// TwinCAT 3 PLC project IDPLC
// ProgramVersion: 3.1.4024.12
// libraries:
//   Tc2_Drive, * (Beckhoff Automation GmbH)
//   Tc2_EtherCAT, * (Beckhoff Automation GmbH)
//   Tc2_Math, * (Beckhoff Automation GmbH)
//   Tc2_MC2, * (Beckhoff Automation GmbH)
//   Tc2_NC, * (Beckhoff Automation GmbH)
//   Tc2_NcDrive, * (Beckhoff Automation GmbH)
//   Tc2_SerialCom, * (Beckhoff Automation GmbH)
//   Tc2_Standard, * (Beckhoff Automation GmbH)
//   Tc2_System, * (Beckhoff Automation GmbH)
//   Tc2_Utilities, * (Beckhoff Automation GmbH)
//   Tc3_Module, * (Beckhoff Automation GmbH)
// project tree:
//   DUTs/ DUT_SENSOR_DATAS_1.TcDUT (not stored), DUT_SENSOR_DATAS_8.TcDUT (not stored), DUT_SENSOR_DATAS_2.TcDUT (not stored), DUT_SENSOR_DATAS_3.TcDUT (not stored), DUT_SENSOR_DATAS_4.TcDUT (not stored), DUT_SENSOR_DATAS_5.TcDUT (not stored), DUT_SENSOR_DATAS_6.TcDUT (not stored), DUT_SENSOR_DATAS_7.TcDUT (not stored), Struct_M_Compensation.TcDUT, ST_P180.TcDUT, ST_P182.TcDUT, ST_P183.TcDUT
//   GVLs/ Global_Variables.TcGVL, Variable_Configuration.TcGVL (not stored)
//   / PlcTask.TcTTO (not stored), RecipeManager.TcRMO (not stored)
//   POUs/0.UserMode/ F_GetSysTime.TcPOU (not stored), UserMode.TcPOU
//   POUs/CommonFB/ExternFB/ FB_LedShow.TcPOU (not stored), FB_PlcEmergencyStop.TcPOU (not stored)
//   POUs/CommonFB/MainFB/ FB_Move.TcPOU, FB_Power.TcPOU, FB_SetAxisPosition.TcPOU, FB_SetMotorAxisPosition.TcPOU, FB_Stop.TcPOU
//   POUs/ MAIN.TcPOU
//   POUs/RS232/ BackgroundEL.TcPOU (not stored), FB_SerialCom.TcPOU (not stored)

// ---- DUTs/Struct_M_Compensation.TcDUT
TYPE Struct_M_Compensation :
STRUCT
	Gap:LREAL;
	PhaseShifterLin:LREAL;
	InRange:BOOL;
END_STRUCT
END_TYPE

// ---- DUTs/ST_P180.TcDUT
//Feedback 2 type
TYPE ST_P180 :
STRUCT
	iActual_lenght:UINT:=224;
	iMax_lenght:UINT:=224;

	Manufacturer:UINT:=2;
	Feedback_type:UINT:=1;
	Feedback_type_string:STRING(29):='hallo';
	Feedback_use:UINT:=3;
	Feedback_direction:UINT:=1;
	(*rsvd*)
		rsvd1:ARRAY[0..2] OF UINT;

	(*Powersettlings*)
		Control_voltage:UINT;
		Wait_time_after_power_up:UINT;
		Connector:UINT;
		rsvd2:ARRAY[0..2] OF UINT;

	(*Process channel*)
		Process_interface:UINT;
		Conector2:UINT;
			(*rsvd*)
				rsvd3:ARRAY[0..1] OF UINT;
			(*Data*)
				(*Sin/Cos*)
					Resulution_per_rotation:UDINT;
					Length_per_signal_period:UDINT;
					Sin_gain_correction:UINT;
					Sin_offset_correction:UINT;
					Cos_gain_correction:UINT;
					Cos_offset_correction:UINT;
					Sin_Cos_1Vss_monitoring:UINT;
					rsvd4:ARRAY[0..10] OF UINT;
				(*TTL*)
					(*Resolution_per_rotation:UDINT;
					Length_per_signal_period:UDINT;
					rsvd5:ARRAY[0..15] OF UINT;*)
				(*Resolver*)
					(*Control_word:UINT;
					Number_of_poles:USINT;
					Exibition_frequency:USINT;
					Transformation_ratio:UINT;
					Phase_shift:UINT;
					Sin_cos_amplitude_monitoring:UINT;
					rsvd6:UINT;
					Amplitude_monitoring_max_limit:UINT;
					Amplitude_monitoring_min_limit:UINT;
					Observer_bandwidth:UINT;
					Observer_correction_factor_Iq_to_acc:UINT;
					rsvd7:ARRAY[0..4] OF UDINT;*)
				(*MES*)
					(*Control_word:UINT;
					rsvd8:UINT;
					sin_offset:UINT;
					cos_offset:UINT;
					Sin_cos_Amplitude_correction:UINT;
					rsvd9:UINT;
					Amplitude_monitoring_max_limit:UINT;
					Amplitude_monitoring_min_limit:UINT;
					Observer_bandwidth:UINT;
					Observer_correction_factor_Iq_to_acc:UINT;
					rsvd10:ARRAY[0..4] OF UDINT;*)
				(*HTL*)
					(*Resulution_per_rotation:UDINT;
					Length_per_signal_period:UDINT;
					rsvd11:ARRAY[0..15] OF UINT;*)
	(*Parameter channel*)
		Parameter_interface:UINT;
		Conector3:UINT;
		Identifier:UDINT;
		Bit_resolution_singelturn_position:UINT;
		Bit_resolution_multiturn_position:UINT;
		Number_of_clockcycles_to_get_singelturn_position:UINT;
		Number_of_clockcycles_to_get_multiturn_position:UINT;
		Digital_name_plate:UINT;
		commutation_mode_adjustable_commutation_offset:UINT;
		Linear_reselution_about_digital_interface_in_nm:UDINT;
		rsvd12:ARRAY[0..3] OF UINT;
		data:ARRAY[0..29] OF UINT;
	(*manufacturer limits settings*)
		Maximum_continous_operation_speed:UINT;
		Maximum_continous_mechenical_speed:UINT;
		Maximum_temperature:UINT;
		rsvd13:ARRAY[0..2] OF UINT;

	FeedbackOption :UDINT:=1;
	Reserve :ARRAY[0..5] OF UINT;
END_STRUCT
END_TYPE

// ---- DUTs/ST_P182.TcDUT
// Feedback 2 gear numerator
TYPE ST_P182 :
STRUCT
	Feedback_2_geat_numerator:UDINT;
END_STRUCT
END_TYPE

// ---- DUTs/ST_P183.TcDUT
// Feedback 2 gear denominator
TYPE ST_P183 :
STRUCT
	Feedback_2_geat_denominator:UDINT;
END_STRUCT
END_TYPE

// ---- GVLs/Global_Variables.TcGVL
//{attribute 'Tc2GvlVarNames'}
VAR_GLOBAL
(*IDControl Ready*)
	IDControlReady:BOOL;
(*RecipeDescription*)
	RecipeSavedDate:STRING;
	RecipeDescription:STRING;
(*Reset*)
	btn_Reset:BOOL;
(*Error Massage*)
	Error:BOOL;
	ErrorID:DINT;
	ErrorDescription:STRING;
(*加载配方参数*)
	LoadRecipeParameters:BOOL;
	loadParametersDone:BOOL;
(*Max Velocity Global*)
	MaxVelocityGlobalVelocity : LREAL;
(*设置光栅bias done *)	
	PositionBiasDone:BOOL;
(*回程差*)
	HysteresisError:LREAL;
(*Drive Status*)
	DriveStatus:DINT;//1:Drive Ready;2:Axis is in operation;0:Others
(*光栅漂移误差阈值*)
	LEDriftErrorThreshold:LREAL:=0.001;
(*Lag Distance threshold*)
	PosDiff_PhaseShifterLin:LREAL:=0.5;
(*key Command*)
	btn_Power:BOOL;
	btn_PowerOn: BOOL;
	btn_PowerOff: BOOL;
(*Compensation Value*)
	M_Compensation:ARRAY[1..18] OF Struct_M_Compensation
:=[
(Gap:=0,		PhaseShifterLin:=0,		InRange:=FALSE),
(Gap:=60,		PhaseShifterLin:=60,	InRange:=FALSE),
(Gap:=68,		PhaseShifterLin:=68,	InRange:=FALSE),
(Gap:=70,		PhaseShifterLin:=70,	InRange:=FALSE),
(Gap:=80,		PhaseShifterLin:=80,	InRange:=FALSE),
(Gap:=90,		PhaseShifterLin:=90,	InRange:=FALSE),
(Gap:=100,		PhaseShifterLin:=100,	InRange:=FALSE),
(Gap:=120,		PhaseShifterLin:=120,	InRange:=FALSE),
(Gap:=140,		PhaseShifterLin:=140,	InRange:=FALSE),
(Gap:=160,		PhaseShifterLin:=160,	InRange:=FALSE),
(Gap:=170,		PhaseShifterLin:=170,	InRange:=FALSE),
(Gap:=180,		PhaseShifterLin:=180,	InRange:=FALSE),
(Gap:=190,		PhaseShifterLin:=190,	InRange:=FALSE),
(Gap:=200,		PhaseShifterLin:=200,	InRange:=FALSE),
(Gap:=210,		PhaseShifterLin:=210,	InRange:=FALSE),
(Gap:=220,		PhaseShifterLin:=220,	InRange:=FALSE),
(Gap:=230,		PhaseShifterLin:=230,	InRange:=FALSE),
(Gap:=3000.001,	PhaseShifterLin:=3000.001,	InRange:=FALSE)];

(*simulation OR NOT*)
	simulation:BOOL;
(*USELinearEncoeder*)
	USELinearEncoder:BOOL:=TRUE;
(*restartTwinCAT*)
	m_restartTC:BOOL;
(*Plc_EmergencyStop *)
	Plc_EmergencyStop  AT %Q*:BOOL:=TRUE;
(*硬急停*)
	Hardware_EmergencyStop :BOOL:=TRUE;
(*LED*)
	Led_Run  AT %Q*:BOOL;
	Led_Error  AT %Q*:BOOL;
(*LimitSwitch*)
	LS_TopFar  :BOOL;
	LS_TopNear  :BOOL;
	LS_BottomFar  :BOOL;//not used
	LS_BottomNear  :BOOL;//not used
	Unreach_LS_Far:BOOL;
	Unreach_LS_Near:BOOL;
(*kill switch*)
	KS_TopFar_Contact1:BOOL;
	KS_TopFar_Contact2:BOOL;
	KS_TopNear_Contact1:BOOL;
	KS_TopNear_Contact2:BOOL;
	KS_BottomFar_Contact1:BOOL;//not used
	KS_BottomFar_Contact2:BOOL;//not used
	KS_BottomNear_Contact1:BOOL;//not used
	KS_BottomNear_Contact2:BOOL;//not used
	
(*E-STOP*)
	KS_CabinetEmergency_contact1:BOOL;
	KS_CabinetEmergency_contact2:BOOL;
	KS_handEmergency1_Contact1:BOOL;
	KS_handEmergency1_Contact2:BOOL;
	KS_handEmergency2_Contact1:BOOL;
	KS_handEmergency2_Contact2:BOOL;
	KS_softEmergency2_Contact:BOOL;

(*aixs_ref*)
	PhaseShifterLin: axis_ref;
(*aixs_ref-motor*)
	PhaseShifterMotor: axis_ref;
(*axis Position*)
	Pos_PhaseShifterLin: LREAL;
(*axis Position-motor*)
	Pos_PhaseShifterMotor: LREAL;
(*axis Position-Delta*)
	DeltaPos_PhaseShifter: LREAL;
(*axis Position-Threshold*)
	ThresholdDeltaPos_PhaseShifter: LREAL:=0.2;
(*axis Velocity*)
	Velo_PhaseShifterLin: LREAL;
(*axis Velocity-motor*)
	Velo_PhaseShifterMotor: LREAL;
(*axis Velocity-Delta*)
	DeltaVelo_PhaseShifter: LREAL;
(*axis Velocity-ThresholdDelta*)
	ThresholdDeltaVelo_PhaseShifter: LREAL:=0.1;
(*axis Torque-motor*)
	Torque_PhaseShifterLin: LREAL;
(*axis Torque-motor*)
	Torque_PhaseShifterMotor: LREAL;
(*axis Torque-Delta*)
	DeltaTorque_PhaseShifter: LREAL;
(*Lag Distance*)
	PosDiff_PhaseShifterLin_actual: LREAL;
(*Lag Distance-Motor*)
	PosDiff_PhaseShifterMotor_actual: LREAL;
(*Delta LagDistance*)
	DeltaPosDiff_PhaseShifter_actual: LREAL;

(***********************Power status and couple statatus***********************)
	st_Power:BOOL;
(************************FB***********************)
	FB_Power:FB_Power;
	FB_PlcEmergencyStop: FB_PlcEmergencyStop;
	FB_Move:FB_Move;
	FB_Stop:FB_Stop;
(********************²¹³¥GapÄ£Ê½£¬µ¥Öá²¹³¥Êý¾Ý************************)
	(*ÊÇ·ñ²¹³¥*)
	USE_SingleAxis_Compensation:BOOL:=TRUE;

	M_CompensationNumber:INT;
	M_DisplayNumber:INT;
	(*Conpensation Position Target*)
	PhaseShifterLinPositionNew:LREAL;

	(*考虑到回程差后，运动到临时位置*)
	PhaseShifterLinPositionNew_temporary :LREAL;
	(*Display Position*)
	PhaseShifterLinPositionDisplay:LREAL;
	(*Display Velocity*)
	PhaseShifterLinVelocityDisplay:LREAL;
	//
	moveStatusPhaseShifterLin: BOOL;
	//
	moveStatusPhaseShifterMotor: BOOL;

(******RS232************)
	RxBufferEL			: ComBuffer;	(* Receive data buffer; used with all receive function blocks *)
	TxBufferEL			: ComBuffer;	(* Transmit data buffer; used with all receive function blocks *)
(*input protection*)
	//
	min_UserGapPositionNew:LREAL:=10;
	max_UserGapPositionNew:LREAL:=200;
	inRange_UserGapPositionNew:BOOL;
		//LE protection position
	min_UserLEProtectionGapPosition:LREAL;
	min_ThresholdGapSoft2LEProtection:LREAL;
	max_UserLEProtectionGapPosition:LREAL;
	max_ThresholdGapSoft2LEProtection:LREAL;
	//
	min_UserGapVelocityNew:LREAL:=0;
	max_UserGapVelocityNew:LREAL:=3;
	inRange_UserGapVelocityNew:BOOL;
	//
	min_UserTaperPositionNew: LREAL:=0;;
	max_UserTaperPositionNew: LREAL:=4;
	inRange_UserTaperPositionNew: BOOL;
	//
	min_UserTaperVelocityNew: LREAL:=0;
	max_UserTaperVelocityNew: LREAL:=1;
	inRange_UserTaperVelocityNew: BOOL;
	
END_VAR

// ---- POUs/CommonFB/MainFB/FB_Power.TcPOU
(****************************************************************
NAME:			FB_PowerOn
DATA:			2017.2.16
VERSION:		1.0.0
DESCRIPTION:	FB_PowerOn
HISTORY:
				2017.2.16		NEW

***************************************************************)
FUNCTION_BLOCK FB_Power
VAR_INPUT
	On:BOOL;
	Off:BOOL;
	Check:BOOL;
END_VAR
VAR_OUTPUT
	FbID:DINT:=1001;
	OnState:DINT;
	OffState: INT;
	OnBusy:BOOL;
	OffBusy:BOOL;
	OnStatus:BOOL;
	OffStatus: BOOL;
	Error:BOOL;
	ErrorID:DINT;
	PowerState:BOOL;
END_VAR
VAR
	PhaseShifterLin_MC_Power: MC_Power;
	fb_ton:TON;
END_VAR

(*power on *)
IF On AND NOT Off THEN
	A_PowerOn();
(*Power Off *)
ELSIF Off AND NOT On THEN
	A_PowerOff();
END_IF
(*Check*)
IF Check THEN
	A_CheckPowerStatus();
END_IF

ACTION A_CheckPowerStatus:
A_PowerMC();
IF  PhaseShifterLin_MC_Power.Status THEN
	PowerState:=1;
ELSIF NOT PhaseShifterLin_MC_Power.Status THEN
	PowerState:=0;
ELSE
	PowerState:=0;
	Error:=TRUE;
	ErrorID:=77;
	(*FB_PlcEmergencyStop();*)
END_IF
END_ACTION

ACTION A_PowerMC:
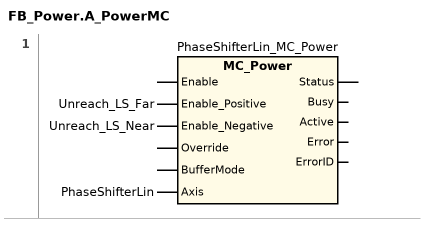
// NETWORK 1
PhaseShifterLin_MC_Power(
    Enable_Positive := Unreach_LS_Far,
    Enable_Negative := Unreach_LS_Near,
    Axis := PhaseShifterLin); // MC_Power
END_ACTION

ACTION A_PowerOff:
OffBusy:=TRUE;
CASE OffState OF
	0:
		IF NOT PhaseShifterLin_MC_Power.Status THEN	(*¶¼Ã»ÉÏµç*)
			OffState:=88;
		ELSE
			OffState:=1;
		END_IF
	1:
		PhaseShifterLin_MC_Power.Enable:=FALSE;
		A_PowerMC();
		OffState:=2;
	2:
		IF NOT PhaseShifterLin_MC_Power.Status THEN	(*¶¼Ã»ÉÏµç*)
			OffState:=88;
		ELSE
			ErrorId:=11;
			OffState:=-100;
		END_IF
	88:
		Off:=FALSE;
		OffState:=0;
		OffBusy:=FALSE;
		OnStatus:=FALSE;
		OffStatus:=TRUE;
		Error:=FALSE;
		ErrorID:=0;
	-100:
		FB_PlcEmergencyStop();
		Off:=FALSE;
		OffState:=-100;
		OffBusy:=FALSE;
		OffStatus:=FALSE;
		Error:=TRUE;

END_CASE
END_ACTION

ACTION A_PowerOn:
OnBusy:=TRUE;
fb_ton(PT:=t#0.5s);
CASE OnState OF
	0:	(*Check*)
		A_PowerMC();
		IF PhaseShifterLin_MC_Power.Error OR NOT PhaseShifterLin_MC_Power.Active THEN		(*FB Error*)
			ErrorID:=1;
			OnState:=99;
		ELSIF PhaseShifterLin_MC_Power.Status THEN		(*ÖáÒÑ¾­¶¼PowerOn£¬²»·ûºÏ¹¦ÄÜ¿éµ÷ÓÃÌõ¼þ*)
			ErrorID:=2;
			OnState:=-100;
		ELSIF NOT PhaseShifterLin_MC_Power.Status THEN		(*Öá¶¼Ã»ÓÐPower£¬×ªÏÂÒ»²½*)
			OnState:=1;
		ELSE
			ErrorID:=3;
			OnState:=-100;
		END_IF
	1:	(*Execute*)
		IF NOT PhaseShifterLin_MC_Power.Status THEN		(*ÔÙ¼ì²é£¬Öá¶¼Ã»ÓÐPower*)
			PhaseShifterLin_MC_Power.Enable:=TRUE;
			A_PowerMC();
			fb_ton.IN:=TRUE;
			OnState:=2;
		ELSE
			ErrorID:=4;
			OnState:=-100;
		END_IF
	2:	(*Wait*)
		A_PowerMC();
		IF NOT PhaseShifterLin_MC_Power.Status THEN		(*Power StatusÐÅºÅ²»µ½£¬¼ÌÐøµÈ´ý£¬Èç¹û³¬Ê±ÔòFB Error*)
			IF NOT fb_ton.Q THEN
				OnState:=2;
			ELSE
				ErrorID:=8;
				OnState:=99;
			END_IF
		ELSIF  PhaseShifterLin_MC_Power.Status THEN			(*ÕýÈ·µç»úÉÏµã×´Ì¬£¬×ªÏÂÒ»²½*)
				OnState:=88;
		ELSE
				ErrorID:=9;
				OnState:=-100;
		END_IF
	88:
		On:=FALSE;
		OnState:=0;
		OnBusy:=FALSE;
		OnStatus:=TRUE;
		OffStatus:=FALSE;
		Error:=FALSE;
		ErrorID:=0;
		fb_ton.IN:=FALSE;
	99:
		On:=FALSE;
		OnState:=99;
		OnBusy:=FALSE;
		OnStatus:=FALSE;
		Error:=TRUE;
		PhaseShifterLin_MC_Power.Enable:=FALSE;
		fb_ton.IN:=FALSE;
	-100:
		FB_PlcEmergencyStop();
		On:=FALSE;
		OnState:=-100;
		OnBusy:=FALSE;
		OnStatus:=FALSE;
		Error:=TRUE;
		PhaseShifterLin_MC_Power.Enable:=FALSE;
		fb_ton.IN:=FALSE;

END_CASE
END_ACTION

END_FUNCTION_BLOCK

// ---- POUs/CommonFB/MainFB/FB_Move.TcPOU
(****************************************************************
NAME:			FB_Move
DATA:			2017.2.17
VERSION:		1.0.0
DESCRIPTION:	FB_Move
HISTORY:
				2017.2.17		NEW
				2018.1.9		ÐÂÔöBCGapMode
***************************************************************)
FUNCTION_BLOCK FB_Move
VAR_INPUT
	(*È«¾Ö*)
	Mode:DINT;
	PowerState:BOOL;
	(*BCGapMode*)
	TargetGapPosition:LREAL;
	TargetGapVelocity:LREAL;
	BCGapMove:BOOL;
	BCGapReset:BOOL;
END_VAR
VAR_OUTPUT
	FbID:DINT:=1001;

	BCGapState:DINT;
	BCGapBusy:BOOL;
	BCGapDone:BOOL;
	GapMoving:BOOL;
	Error:BOOL;
	ErrorID:DINT;
END_VAR
VAR
	PhaseShifterLin_MC_MoveAbsolute: MC_MoveAbsolute;
	fb_ton: TON;
	fb_ton1: TON;
	fb_ton2: TON;
	fb_ton_debug_1:TON;
	fb_ton_debug_2:TON;
	fb_ton_debug_3:TON;
	fb_ton_debug_4:TON;
	fb_ton_BC:TON;
	fb_ton_BC_2:TON;
	
END_VAR

IF PowerState=1 THEN
	IF Mode=1 AND BCGapMove THEN
		A_BCGapMove();
	END_IF
END_IF

ACTION A_BCGapMove:
IF BCGapMove THEN
	BCGapBusy:=TRUE;
	BCGapDone:=FALSE;
	fb_ton_BC(PT:=t#80s);(*2mm/s max spees,120mmÐÐ³Ì£¬60sÄÚ×ßÍê*)
	A_MoveMC();
	IF  PhaseShifterLin.Status.Moving  THEN
		GapMoving:=TRUE;
	ELSE
		GapMoving:=FALSE;
	END_IF
	CASE BCGapState OF
		0:
			IF PhaseShifterLin.Status.Moving THEN	(*ÖáÕýÔÚÔËÐÐ£¬Ñ­»·¸Ã²½µÈ´ý*)
				BCGapState:=88;
			ELSIF PhaseShifterLin.Status.NotMoving THEN	(*Öá¶¼´¦ÓÚÍ£Ö¹×´Ì¬Ê±£¬×ªÏÂÒ»²½*)
				BCGapState:=1;
			END_IF
		1:
			PhaseShifterLin_MC_MoveAbsolute.Position:=TargetGapPosition;
			PhaseShifterLin_MC_MoveAbsolute.Velocity:=TargetGapVelocity;
			PhaseShifterLin_MC_MoveAbsolute.Execute:=TRUE;
			fb_ton_BC.IN:=TRUE;
			BCGapState:=2;
		2:
			IF NOT PhaseShifterLin_MC_MoveAbsolute.Done THEN		(*ÔË¶¯ÖÐ£¬¼ì²éDoneÐÅºÅ£¬Ã»ÓÐÔòÑ­»·*)
				BCGapState:=2;
			ELSIF PhaseShifterLin_MC_MoveAbsolute.Done THEN		(*ÔË¶¯Íê³É£¬×ªÏÂÒ»²½*)
				BCGapState:=88;
			END_IF
	
		88:
			BCGapMove:=FALSE;
			BCGapState:=0;
			BCGapBusy:=FALSE;
			BCGapDone:=TRUE;
			Error:=FALSE;
			ErrorID:=0;
			PhaseShifterLin_MC_MoveAbsolute.Execute:=FALSE;
			fb_ton_BC.IN:=FALSE;
		89:
			BCGapMove:=FALSE;
			BCGapState:=0;
			BCGapBusy:=FALSE;
			BCGapDone:=FALSE;
			Error:=FALSE;
			ErrorID:=0;
			PhaseShifterLin_MC_MoveAbsolute.Execute:=FALSE;
			fb_ton_BC.IN:=FALSE;
		99:
			BCGapMove:=FALSE;
			BCGapState:=99;
			BCGapBusy:=FALSE;
			BCGapDone:=FALSE;
			Error:=TRUE;
			PhaseShifterLin_MC_MoveAbsolute.Execute:=FALSE;
			fb_ton_BC.IN:=FALSE;
		-100:
			FB_PlcEmergencyStop();
			BCGapMove:=FALSE;
			BCGapState:=-100;
			BCGapBusy:=FALSE;
			BCGapDone:=FALSE;
			Error:=TRUE;
			PhaseShifterLin_MC_MoveAbsolute.Execute:=FALSE;
			fb_ton_BC.IN:=FALSE;
	END_CASE
	IF BCGapReset THEN
		BCGapReset:=FALSE;
		BCGapMove:=FALSE;
		BCGapState:=0;
		BCGapBusy:=FALSE;
		BCGapDone:=FALSE;
		Error:=FALSE;
		ErrorID:=0;
		PhaseShifterLin_MC_MoveAbsolute.Execute:=FALSE;
		fb_ton_BC.IN:=FALSE;
	END_IF
END_IF
END_ACTION

ACTION A_MoveMC:
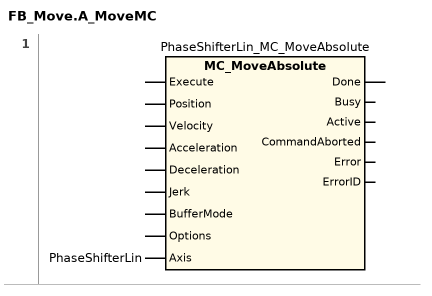
// NETWORK 1
PhaseShifterLin_MC_MoveAbsolute(Axis := PhaseShifterLin); // MC_MoveAbsolute
END_ACTION

END_FUNCTION_BLOCK

// ---- POUs/CommonFB/MainFB/FB_Stop.TcPOU
FUNCTION_BLOCK FB_Stop
VAR_INPUT
(*È«¾Ö*)
	Mode:DINT;
	PowerState:BOOL;
	(*BCGapMode*)
	BCGapStop:BOOL;
END_VAR
VAR_OUTPUT
	FbID:DINT:=1001;

	BCGapState:DINT;
	BCGapBusy:BOOL;
	BCGapDone:BOOL;

	Error:BOOL;
	ErrorID:DINT;
END_VAR
VAR
	PhaseShifterLin_MC_Stop: MC_Stop;
	fb_ton: TON;
	fb_ton1: TON;
	fb_ton2: TON;
	fb_ton_debug_1:TON;
	fb_ton_debug_2:TON;
	fb_ton_debug_3:TON;
	fb_ton_debug_4:TON;
	fb_ton_BC: TON;

END_VAR

IF PowerState=1 THEN
	IF Mode=1 AND BCGapStop THEN
		A_BCGapStop();
	ELSE
		FB_PlcEmergencyStop();
	END_IF
END_IF

ACTION A_BCGapStop:
IF BCGapStop THEN
BCGapBusy:=TRUE;
BCGapDone:=FALSE;
fb_ton_BC(PT:=t#100ms);
A_StopMC();
CASE BCGapState OF
	0:
		IF PhaseShifterLin_MC_Stop.Error  THEN
			ErrorID:=1;
			BCGapState:=-100;
			PhaseShifterLin_MC_Stop.Execute:=FALSE;
			A_StopMC();
		ELSE
			BCGapState:=1;
		END_IF
	1:
		PhaseShifterLin_MC_Stop.Execute:=TRUE;
		fb_ton_BC.IN:=TRUE;
		BCGapState:=2;
	2:
		IF  NOT PhaseShifterLin_MC_Stop.Done  THEN
				BCGapState:=2;
		ELSE
			BCGapState:=88;
			PhaseShifterLin_MC_Stop.Execute:=FALSE;
			A_StopMC();
		END_IF

	88:
		BCGapStop:=FALSE;
		BCGapState:=0;
		BCGapBusy:=FALSE;
		BCGapDone:=TRUE;
		Error:=FALSE;
		ErrorID:=0;
		fb_ton_BC.IN:=FALSE;

	-100:
		FB_PlcEmergencyStop();
		BCGapStop:=FALSE;
		BCGapState:=-100;
		BCGapBusy:=FALSE;
		BCGapDone:=FALSE;
		Error:=TRUE;
		PhaseShifterLin_MC_Stop.Execute:=FALSE;
		A_StopMC();
		fb_ton_BC.IN:=FALSE;

END_CASE
END_IF
END_ACTION

ACTION A_StopMC:
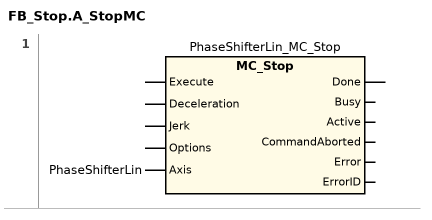
// NETWORK 1
PhaseShifterLin_MC_Stop(Axis := PhaseShifterLin); // MC_Stop
END_ACTION

END_FUNCTION_BLOCK

// ---- POUs/0.UserMode/UserMode.TcPOU
PROGRAM UserMode
VAR

(*GapMode*)
	UserGapPositionNew:LREAL:=20;//target
	UserGapVelocityNew:LREAL:=1;//target
	UserGapPositionDisplay:LREAL;//current
	UserGapVelocityDisplay:LREAL;//current
	//
	(**)
	btn_UserGapMove:BOOL;
	btn_UserGapStop:BOOL;
	(*Var*)
	fb_ton1:TON;
	fb_ton2:TON;
	fb_ton3:TON;
	(*Status*)
	State:DINT;
	Busy:BOOL;
	InitPowerDone:BOOL;
	InitCompensationDatasDone:BOOL;
	(*FB*)
	m_state: DINT;
	n_state: DINT;
	s_state: DINT;
	(*¼ì²âµ½ÏÞÎ»£¬»Ö¸´Move×´Ì¬*)
	FTrig_ReachLS: F_TRIG;
	FTrig_btn_GapMove: F_TRIG;
	GapOutRange: BOOL;
	(*PowerOff*)
	d_state: DINT;
	i: INT;
	j: INT;
	k: INT;
	moni_State:DINT;
	TargetPosLessThanCurrentPos:BOOL;
	PositiveMoving:BOOL;
	HysteresisMoving:BOOL;
	NoneHysteresisMoving:BOOL;
	(*Spectroscopy scanning Mode*)
	IsSSMotionMode:BOOL;
	RegularMotionMode:BOOL;
	SSMotionMode:BOOL;
	SS_StepSize:LREAL:=0.001;
	SS_StepNumber:INT:=10;
	SS_StepVelocity:LREAL:=1;
	SS_Move:BOOL;
	SS_Stop:BOOL;
	SS_MoveState:DINT;
	SS_StopState:DINT;
	SS_currentStep:DINT:=0;
	SS_StepSystemTime_Begin:ARRAY[0..100] OF ULINT;
	SS_StepSystemTime_End:ARRAY[0..100] OF ULINT;
	SS_StepCountTime:ARRAY[0..100] OF ULINT;
	SS_TimeCountBegin:BOOL;
	m: INT;
	SS_TON: TON;
	StepEachTime:TIME;
	StepEachTime_ms:INT:=1000;//ms
	SS_OTSTRUCT :OTSTRUCT ;
	SS_StartPositionDisplay:LREAL;
	RTRG_SS_StartPositionDisplay:R_TRIG;
	SS_InitStartPositionDone:BOOL;
	
	//
	min_SS_StepSize	: LREAL:=0;
	max_SS_StepSize	: LREAL:=200;
	inRange_SS_StepSize	: BOOL;
	//
	min_SS_StepNumber	: INT:=1;
	max_SS_StepNumber	: INT:=1000;
	inRange_SS_StepNumber	: BOOL;
	//
	min_SS_StepVelocity:LREAL:=0;
	max_SS_StepVelocity:LREAL:=1;
	inRange_SS_StepVelocity:BOOL;
	//
	min_StepEachTime_ms:INT:=100;
	max_StepEachTime_ms:INT:=10000;
	inRange_StepEachTime_ms:BOOL;
	l: INT;
	testa: BOOL;
	testb: BOOL;
	Threshold_GapChangeFlag: LREAL;
	Threshold_TaperChangeFlag: LREAL;
	TaperAndGapSafetyfactor: LREAL:=1;
	
		//
	//Global Chain protection-MPS
	Global_ChainProtection_MPS_StorageRingReady:BOOL;
	Global_ChainProtection_MPS_On: BOOL;
	Global_ChainProtection_MPS_MaxGapValue: LREAL;
	Global_ChainProtection_MPS_MoveVelocity: LREAL;
	Global_ChainProtection_MPS_Done: BOOL;
	//Global_ChainProtection_Error: BOOL;
	//Global_ChainProtection_ErrorID: INT;
	//Global_ChainProtection_ErrorDescription: STRING;
	Global_ChainProtection_MPS_ManualOperation:BOOL:=TRUE;
	Global_ChainProtection_MPS_FTRIG:F_TRIG;
	Global_ChainProtection_MPS_FTRIG_Manul:F_TRIG;
	Global_ChainProtection_MPS_TON:TON;
	Global_ChainProtection_MPS_Triggered:BOOL;
	Global_ChainProtection_MPS_In:BOOL;
	Global_ChainProtection_MPS_In1 AT%I* :BOOL;//下降沿表示触发
	Global_ChainProtection_MPS_In2 AT%I* :BOOL;
	Global_ChainProtection_MPS_State:DINT;
	Global_ChainProtection_MPS_Out1 AT%Q* :BOOL;//上升沿标识到达最大间隙，连锁保护成功
	Global_ChainProtection_MPS_Out2 AT%Q* :BOOL;
	Global_ChainProtection_MPS_TON_Stop2Move:TON;
	Global_ChainProtection_MPS_TON_Stop2Move_InTaperMode:TON;
	Global_ChainProtection_MPS_TON_Power2Move:TON;
	//Global Chain protection-EPS
	Global_ChainProtection_EPS_BeamLineReady:BOOL;
	Global_ChainProtection_EPS_On: BOOL;
	Global_ChainProtection_EPS_MaxGapValue: LREAL;
	Global_ChainProtection_EPS_MoveVelocity: LREAL;
	Global_ChainProtection_EPS_Done: BOOL;
	//Global_ChainProtection_Error: BOOL;
	//Global_ChainProtection_ErrorID: INT;
	//Global_ChainProtection_ErrorDescription: STRING;
	Global_ChainProtection_EPS_ManualOperation:BOOL:=TRUE;
	Global_ChainProtection_EPS_FTRIG:F_TRIG;
	Global_ChainProtection_EPS_FTRIG_Manul:F_TRIG;
	Global_ChainProtection_EPS_TON:TON;
	Global_ChainProtection_EPS_Triggered:BOOL;
	Global_ChainProtection_EPS_In:BOOL;
	Global_ChainProtection_EPS_In1 AT%I* :BOOL;//下降沿表示触发
	Global_ChainProtection_EPS_In2 AT%I* :BOOL;
	Global_ChainProtection_EPS_State:DINT;
	Global_ChainProtection_EPS_Out1 AT%Q* :BOOL;//上升沿标识到达最大间隙，连锁保护成功
	Global_ChainProtection_EPS_Out2 AT%Q* :BOOL;
	Global_ChainProtection_EPS_TON_Stop2Move:TON;
	Global_ChainProtection_EPS_TON_Stop2Move_InTaperMode:TON;
	Global_ChainProtection_EPS_TON_Power2Move:TON;
	//
	Threshold_motorsTargetPosCalculate:LREAL;
	
	PhaseShifterLinPositionNewTemp: LREAL;
		//OneKeyToMaxGap
	btn_OneKeyToMaxGap:BOOL;
	OneKeyToMaxGap_RTRIG:R_TRIG;
	OneKeyToMaxGap_TON:TON;
	OneKeyToMaxGap_Triggered:BOOL;
	OneKeyToMaxGap_State:DINT;
	OneKeyToMaxGap_TON_Stop2Move:TON;
	OneKeyToMaxGap_TON_Stop2Move_InTaperMode:TON;
	OneKeyToMaxGap_TON_Power2Move:TON;
	OneKeyToMaxGap_Done:BOOL;
END_VAR

IF NOT PositionBiasDone THEN
	RETURN;
END_IF
IF NOT loadParametersDone THEN
	RETURN;
END_IF
(*btn_Power On/Off*)
IF btn_Power AND NOT st_Power THEN
	btn_PowerOn:=TRUE;
	btn_Power:=FALSE;
END_IF
IF btn_Power AND st_Power THEN
	btn_PowerOff:=TRUE;
	btn_Power:=FALSE;
END_IF
IF btn_PowerOn THEN
	A_PowerOn();
END_IF
IF btn_PowerOff THEN
	A_PowerOff();
END_IF


(*补偿数据处理*)
A_InitCompensationData();

(*常规磁间隙开合*)
IF RegularMotionMode AND NOT SSMotionMode THEN
	A_RegularMotion();
END_IF

(*Spectroscopy scanning Mode*)
IF IsSSMotionMode THEN
	SSMotionMode:=TRUE;
	RegularMotionMode:=FALSE;
ELSE
	SSMotionMode:=FALSE;
	RegularMotionMode:=TRUE;
END_IF
IF	SSMotionMode AND NOT RegularMotionMode THEN
	A_SpectroscopyScanningMotion();
END_IF

A_CheckMotorsPos();

(*GlobalChainProtection*)
A_GlobalChainProtection_MPS();
A_GlobalChainProtection_EPS();

(*A_OneKeyToMaxGap*)
A_OneKeyToMaxGap();

ACTION A_CheckMotorsPos:
//
//目标位置速度超出阈值判断
//
//gap posiion
IF UserGapPositionNew<min_UserGapPositionNew OR UserGapPositionNew>max_UserGapPositionNew THEN
	inRange_UserGapPositionNew:=FALSE;
END_IF
IF UserGapPositionNew>=min_UserGapPositionNew AND UserGapPositionNew<=max_UserGapPositionNew THEN
	inRange_UserGapPositionNew:=TRUE;
END_IF
//gap velocity
IF UserGapVelocityNew<min_UserGapVelocityNew OR UserGapVelocityNew>max_UserGapVelocityNew THEN
	inRange_UserGapVelocityNew:=FALSE;
END_IF
IF UserGapVelocityNew>=min_UserGapVelocityNew AND UserGapVelocityNew<=max_UserGapVelocityNew THEN
	inRange_UserGapVelocityNew:=TRUE;
END_IF
//SS Mode
IF SS_StepSize<min_SS_StepSize OR SS_StepSize>max_SS_StepSize THEN
	inRange_SS_StepSize:=FALSE;
END_IF
IF SS_StepSize>=min_SS_StepSize AND SS_StepSize<=max_SS_StepSize THEN
	inRange_SS_StepSize:=TRUE;
END_IF
IF SS_StepNumber<min_SS_StepNumber OR SS_StepNumber>max_SS_StepNumber THEN
	inRange_SS_StepNumber:=FALSE;
END_IF
IF SS_StepNumber>=min_SS_StepNumber AND SS_StepNumber<=max_SS_StepNumber THEN
	inRange_SS_StepNumber:=TRUE;
END_IF
IF SS_StepVelocity<min_SS_StepVelocity OR SS_StepVelocity>max_SS_StepVelocity THEN
	inRange_SS_StepVelocity:=FALSE;
END_IF
IF SS_StepVelocity>=min_SS_StepVelocity AND SS_StepVelocity<=max_SS_StepVelocity THEN
	inRange_SS_StepVelocity:=TRUE;
END_IF
IF StepEachTime_ms<min_StepEachTime_ms OR StepEachTime_ms>max_StepEachTime_ms THEN
	inRange_StepEachTime_ms:=FALSE;
END_IF
IF StepEachTime_ms>=min_StepEachTime_ms AND StepEachTime_ms<=max_StepEachTime_ms THEN
	inRange_StepEachTime_ms:=TRUE;
END_IF


//
//输入速度和位置保护
//
IF btn_UserGapMove  AND NOT SSMotionMode AND RegularMotionMode THEN
	IF NOT inRange_UserGapPositionNew THEN
		btn_UserGapStop:=TRUE;
		btn_UserGapMove:=FALSE;
		Error:=TRUE;
		ErrorId:=801;
		ErrorDescription:='target Gap position out of range,please check';
		RETURN;
	ELSE
		//btn_UserGapStop:=FALSE;
		Error:=FALSE;
		ErrorId:=0;
		ErrorDescription:='';	
	END_IF
	IF NOT inRange_UserGapVelocityNew THEN
		btn_UserGapStop:=TRUE;
		btn_UserGapMove:=FALSE;
		Error:=TRUE;
		ErrorId:=802;
		ErrorDescription:='target Gap velocity out of range,please check';
		RETURN;
	ELSE
		//btn_UserGapStop:=FALSE;
		Error:=FALSE;
		ErrorId:=0;
		ErrorDescription:='';
	END_IF
END_IF

//
//运动过程中，监控目标位置速度
//
IF moveStatusPhaseShifterLin THEN
	IF NOT inRange_UserGapPositionNew THEN
		btn_UserGapStop:=TRUE;
		Error:=TRUE;
		ErrorId:=805;
		ErrorDescription:='target Gap position out of range in moving process!';
		FB_PlcEmergencyStop();
	END_IF
	IF NOT inRange_UserGapVelocityNew THEN
		btn_UserGapStop:=TRUE;
		Error:=TRUE;
		ErrorId:=806;
		ErrorDescription:='target Gap velocity out of range in moving process!';
		FB_PlcEmergencyStop();
	END_IF
END_IF
//
//运动过程中，监控每一个轴的目标位置，目标位置若超出阈值，Emergency
//
IF moveStatusPhaseShifterLin THEN
		IF PhaseShifterLinPositionNew<min_UserGapPositionNew OR PhaseShifterLinPositionNew>max_UserGapPositionNew THEN
			btn_UserGapStop:=TRUE;
			Error:=TRUE;
			ErrorId:=809;
			ErrorDescription:='target PhaseShifterLinPositionNew out of range in moving process!';
			FB_PlcEmergencyStop();
		END_IF
END_IF
END_ACTION

ACTION A_GlobalChainProtection_EPS:
//硬线输入定义
Global_ChainProtection_EPS_In:=Global_ChainProtection_EPS_In1 AND Global_ChainProtection_EPS_In2;
//硬线输出定义
Global_ChainProtection_EPS_Out1:=Global_ChainProtection_EPS_Done;
Global_ChainProtection_EPS_Out2:=Global_ChainProtection_EPS_Done;
//总开关
IF NOT Global_ChainProtection_EPS_On THEN
	RETURN;
END_IF
//判断插入件状态，是否就位
//IF NOT IDControlReady THEN
//	Global_ChainProtection_EPS_Done:=FALSE;
//	Error:= TRUE;
//	ErrorID:= 1501;
//	ErrorDescription:='ID NOT READY!';
//	RETURN;
//END_IF
//判断储存环是否给出就位信号，暂时由参数表给出TRUE，最终将由IOC接受PV
IF 	NOT Global_ChainProtection_EPS_BeamLineReady THEN
	Global_ChainProtection_EPS_Done:=FALSE;
	Error:= TRUE;
	ErrorID:= 1503;
	ErrorDescription:='Global_ChainProtection_EPS_BeamLineReady NOT Ready';
	RETURN;
END_IF
//
//全局连锁保护程序开始
//
//0.检测到下降沿，触发
//1.判断电机是否在开启状态,没有就打开电源
//2.判断是否在Moving状态,若有就Stop
//3.将磁间隙打开到至最大阈值
//4.到位后给出反馈，且安全PLC触发
Global_ChainProtection_EPS_FTRIG(CLK:=Global_ChainProtection_EPS_In);
IF Global_ChainProtection_EPS_FTRIG.Q THEN
	Global_ChainProtection_EPS_Triggered:=TRUE;
END_IF
Global_ChainProtection_EPS_FTRIG_Manul(CLK:=Global_ChainProtection_EPS_ManualOperation);
IF Global_ChainProtection_EPS_FTRIG_Manul.Q THEN
	Global_ChainProtection_EPS_Triggered:=TRUE;
END_IF
IF Global_ChainProtection_EPS_Triggered THEN
	CASE Global_ChainProtection_EPS_State OF
		0://1.判断电机是否在开启状态,没有就打开电源
			IF st_Power=1 THEN
				Global_ChainProtection_EPS_State:=1;
			ELSE
				btn_PowerOn:=TRUE;
				IF btn_PowerOn THEN
					A_PowerOn();
				END_IF
			END_IF
		1://1.判断是否在谱学扫描模式，如果是，则切换回正常运动模式
			IF IsSSMotionMode THEN
				SS_Stop:=TRUE;
				IsSSMotionMode:=FALSE;
			END_IF
			Global_ChainProtection_EPS_State:=2;
		2://判断是否在taper，如果在taper,则判断是否在运动，如果是，则停止运动,0.5sh后，转入下一步
			(*IF TaperOrNot THEN
				IF moveStatusLeftTop OR moveStatusRightTop OR moveStatusLeftBottom OR moveStatusRightBottom THEN
					btn_UserGapStop:=TRUE;
				ELSE
					Global_ChainProtection_EPS_TON_Stop2Move_InTaperMode(PT:=T#0.5S);
					Global_ChainProtection_EPS_TON_Stop2Move_InTaperMode.IN:=TRUE;
					IF Global_ChainProtection_EPS_TON_Stop2Move_InTaperMode.Q THEN
						TaperOrNot:=FALSE;//关闭taper模式
						Global_ChainProtection_EPS_State:=3;
					END_IF
				END_IF
			ELSE
			*)
				Global_ChainProtection_EPS_State:=3;
			//END_IF
		3://3.判断是否在Moving状态,若有就Stop.Taper模式已处理完，此处开始走正常GAP开合逻辑
			IF moveStatusPhaseShifterLin THEN
				btn_UserGapStop:=TRUE;
			ELSE
				Global_ChainProtection_EPS_TON_Stop2Move(PT:=T#0.5S);
				Global_ChainProtection_EPS_TON_Stop2Move.IN:=TRUE;
				IF Global_ChainProtection_EPS_TON_Stop2Move.Q THEN
					Global_ChainProtection_EPS_State:=4;
				END_IF
			END_IF
		4://当前磁间隙如何和最大磁间隙差别不大，不超过0.1，则直接保护
			IF ABS(UserGapPositionDisplay-Global_ChainProtection_EPS_MaxGapValue)<=0.1 THEN
				Global_ChainProtection_EPS_Done:=TRUE;
				Plc_EmergencyStop:=FALSE;	
				Error:=TRUE;
				ErrorID:=1506;
				ErrorDescription:='EPS Triggered,but ABS(UserGapPositionDisplay-Global_ChainProtection_EPS_MaxGapValue)<=0.1 ';	
			ELSE
				Global_ChainProtection_EPS_State:=5;
			END_IF
		5://5.将磁间隙打开到至最大阈值
			Global_ChainProtection_EPS_TON(PT:=INT_TO_TIME(LREAL_TO_INT(Global_ChainProtection_EPS_MaxGapValue/Global_ChainProtection_EPS_MoveVelocity+30))*1000);
			Global_ChainProtection_EPS_TON.IN:=TRUE;
			Global_ChainProtection_EPS_TON_Power2Move(PT:=T#0.1S);
			Global_ChainProtection_EPS_TON_Power2Move.IN:=TRUE;
			UserGapPositionNew:=Global_ChainProtection_EPS_MaxGapValue;
			UserGapVelocityNew:=Global_ChainProtection_EPS_MoveVelocity;
			btn_UserGapMove:=TRUE;
			IF Global_ChainProtection_EPS_TON_Power2Move.Q THEN
				IF FB_MOVE.BCGapDone THEN
					Global_ChainProtection_EPS_State:=88;
				END_IF
			END_IF
			IF Global_ChainProtection_EPS_TON.Q THEN//如果150s后，还没有运动到指定gap，则报错
				Global_ChainProtection_EPS_State:=-100;
			END_IF
		88://4.到位后给出反馈，且安全PLC触发
			Global_ChainProtection_EPS_Done:=TRUE;
			Plc_EmergencyStop:=FALSE;	
			Error:=TRUE;
			ErrorID:=1504;
			ErrorDescription:='Global_ChainProtection_EPS Triggered ';	
		-100:
			Global_ChainProtection_EPS_Done:=FALSE;
			Error:=TRUE;
			ErrorID:=1505;
			ErrorDescription:='NOT MOVING TO MAXGAP';
	END_CASE
END_IF
END_ACTION

ACTION A_GlobalChainProtection_MPS:
//硬线输入定义
Global_ChainProtection_MPS_In:=Global_ChainProtection_MPS_In1 AND Global_ChainProtection_MPS_In2;
//硬线输出定义
Global_ChainProtection_MPS_Out1:=Global_ChainProtection_MPS_Done;
Global_ChainProtection_MPS_Out2:=Global_ChainProtection_MPS_Done;
//总开关
IF NOT Global_ChainProtection_MPS_On THEN
	RETURN;
END_IF
//判断插入件状态，是否就位
//IF NOT IDControlReady THEN
//	Global_ChainProtection_MPS_Done:=FALSE;
//	Error:= TRUE;
//	ErrorID:= 1401;
//	ErrorDescription:='ID NOT READY!';
//	RETURN;
//END_IF
//判断储存环是否给出就位信号，暂时由参数表给出TRUE，最终将由IOC接受PV
IF 	NOT Global_ChainProtection_MPS_StorageRingReady THEN
	Global_ChainProtection_MPS_Done:=FALSE;
	Error:= TRUE;
	ErrorID:= 1403;
	ErrorDescription:='StorageRingChainProtection NOT Ready';
	RETURN;
END_IF
//
//全局连锁保护程序开始
//
//0.检测到下降沿，触发
//1.判断电机是否在开启状态,没有就打开电源
//2.判断是否在Moving状态,若有就Stop
//3.将磁间隙打开到至最大阈值
//4.到位后给出反馈，且安全PLC触发
Global_ChainProtection_MPS_FTRIG(CLK:=Global_ChainProtection_MPS_In);
IF Global_ChainProtection_MPS_FTRIG.Q THEN
	Global_ChainProtection_MPS_Triggered:=TRUE;
END_IF
Global_ChainProtection_MPS_FTRIG_Manul(CLK:=Global_ChainProtection_MPS_ManualOperation);
IF Global_ChainProtection_MPS_FTRIG_Manul.Q THEN
	Global_ChainProtection_MPS_Triggered:=TRUE;
END_IF
IF Global_ChainProtection_MPS_Triggered THEN
	CASE Global_ChainProtection_MPS_State OF
		0://1.判断电机是否在开启状态,没有就打开电源
			IF st_Power=1 THEN
				Global_ChainProtection_MPS_State:=1;
			ELSE
				btn_PowerOn:=TRUE;
				IF btn_PowerOn THEN
					A_PowerOn();
				END_IF
			END_IF
		1://1.判断是否在谱学扫描模式，如果是，则切换回正常运动模式
			IF IsSSMotionMode THEN
				SS_Stop:=TRUE;
				IsSSMotionMode:=FALSE;
			END_IF
			Global_ChainProtection_MPS_State:=2;
		2://判断是否在taper，如果在taper,则判断是否在运动，如果是，则停止运动,0.5sh后，转入下一步
			(*IF TaperOrNot THEN
				IF moveStatusLeftTop OR moveStatusRightTop OR moveStatusLeftBottom OR moveStatusRightBottom THEN
					btn_UserGapStop:=TRUE;
				ELSE
					Global_ChainProtection_MPS_TON_Stop2Move_InTaperMode(PT:=T#0.5S);
					Global_ChainProtection_MPS_TON_Stop2Move_InTaperMode.IN:=TRUE;
					IF Global_ChainProtection_MPS_TON_Stop2Move_InTaperMode.Q THEN
						TaperOrNot:=FALSE;//关闭taper模式
						Global_ChainProtection_MPS_State:=3;
					END_IF
				END_IF
			ELSE
			*)
				Global_ChainProtection_MPS_State:=3;
			//END_IF
		3://3.判断是否在Moving状态,若有就Stop.Taper模式已处理完，此处开始走正常GAP开合逻辑
			IF moveStatusPhaseShifterLin THEN
				btn_UserGapStop:=TRUE;
			ELSE
				Global_ChainProtection_MPS_TON_Stop2Move(PT:=T#0.5S);
				Global_ChainProtection_MPS_TON_Stop2Move.IN:=TRUE;
				IF Global_ChainProtection_MPS_TON_Stop2Move.Q THEN
					Global_ChainProtection_MPS_State:=4;
				END_IF
			END_IF
		4://当前磁间隙如何和最大磁间隙差别不大，不超过0.1，则直接保护
			IF ABS(UserGapPositionDisplay-Global_ChainProtection_MPS_MaxGapValue)<=0.1 THEN
				Global_ChainProtection_MPS_Done:=TRUE;
				Plc_EmergencyStop:=FALSE;	
				Error:=TRUE;
				ErrorID:=1406;
				ErrorDescription:='MPS Triggered,but ABS(UserGapPositionDisplay-Global_ChainProtection_MPS_MaxGapValue)<=0.1 ';	
			ELSE
				Global_ChainProtection_MPS_State:=5;
			END_IF
		5://5.将磁间隙打开到至最大阈值
			Global_ChainProtection_MPS_TON(PT:=INT_TO_TIME(LREAL_TO_INT(Global_ChainProtection_MPS_MaxGapValue/Global_ChainProtection_MPS_MoveVelocity+30))*1000);
			Global_ChainProtection_MPS_TON.IN:=TRUE;
			Global_ChainProtection_MPS_TON_Power2Move(PT:=T#0.1S);
			Global_ChainProtection_MPS_TON_Power2Move.IN:=TRUE;
			UserGapPositionNew:=Global_ChainProtection_MPS_MaxGapValue;
			UserGapVelocityNew:=Global_ChainProtection_MPS_MoveVelocity;
			btn_UserGapMove:=TRUE;
			IF Global_ChainProtection_MPS_TON_Power2Move.Q THEN
				IF FB_MOVE.BCGapDone THEN
					Global_ChainProtection_MPS_State:=88;
				END_IF
			END_IF
			IF Global_ChainProtection_MPS_TON.Q THEN//如果150s后，还没有运动到指定gap，则报错
				Global_ChainProtection_MPS_State:=-100;
			END_IF
		88://4.到位后给出反馈，且安全PLC触发
			Global_ChainProtection_MPS_Done:=TRUE;
			Plc_EmergencyStop:=FALSE;	
			Error:=TRUE;
			ErrorID:=1404;
			ErrorDescription:='Global_ChainProtection_MPS Triggered ';	
		-100:
			Global_ChainProtection_MPS_Done:=FALSE;
			Error:=TRUE;
			ErrorID:=1405;
			ErrorDescription:='NOT MOVING TO MAXGAP';
	END_CASE
END_IF
END_ACTION

ACTION A_InitCompensationData:
(*补偿开始*)
IF USE_SingleAxis_Compensation THEN
	//
	//1.目标位置解算
	//
	//左轴目标位置解算
	FOR	i:= 1 TO 17 DO
			IF UserGapPositionNew<M_Compensation[i+1].Gap AND UserGapPositionNew>=M_Compensation[i].Gap THEN
				IF i<>18 THEN
					PhaseShifterLinPositionNew:=(((UserGapPositionNew-M_Compensation[i].Gap)*(M_Compensation[i+1].PhaseShifterLin-M_Compensation[i].PhaseShifterLin))
							/(M_Compensation[i+1].Gap-M_Compensation[i].Gap))+M_Compensation[i].PhaseShifterLin;
					M_CompensationNumber:=i;
					InitCompensationDatasDone:=TRUE;
				ELSIF i=18 AND UserGapPositionNew=M_Compensation[i].Gap THEN		(*Gap=14µÄÌØÊâÇé¿ö*)
					(**)
					PhaseShifterLinPositionNew:=M_Compensation[i].PhaseShifterLin;
					M_CompensationNumber:=i;
					InitCompensationDatasDone:=TRUE;
				ELSE
					PhaseShifterLinPositionNew:=UserGapPositionNew;
					M_CompensationNumber:=i;
					InitCompensationDatasDone:=TRUE;
				END_IF
			END_IF
	END_FOR

	//显示位置反解算
	FOR k:= 1 TO 17 DO
			IF Pos_PhaseShifterLin<M_Compensation[k+1].PhaseShifterLin AND Pos_PhaseShifterLin>=M_Compensation[k].PhaseShifterLin THEN
				UserGapPositionDisplay:=((Pos_PhaseShifterLin-M_Compensation[k].PhaseShifterLin)*(M_Compensation[k+1].Gap-M_Compensation[k].Gap))
											/(M_Compensation[k+1].PhaseShifterLin-M_Compensation[k].PhaseShifterLin)+M_Compensation[k].Gap;
				UserGapPositionDisplay:=DINT_TO_LREAL(LREAL_TO_DINT(UserGapPositionDisplay*100000))/100000;
			END_IF
	END_FOR
END_IF
(*速度可以不用解算，直接用即可*)
PhaseShifterLinVelocityDisplay:=Velo_PhaseShifterLin;
//Gap velocity
UserGapVelocityDisplay:=DINT_TO_LREAL(LREAL_TO_DINT(PhaseShifterLinVelocityDisplay*100000))/100000;


(*解算单轴位置后，核验并做保护*)
IF ABS(PhaseShifterLinPositionNew-UserGapPositionNew)>Threshold_motorsTargetPosCalculate THEN
	ErrorID:=1601;
	Error:=TRUE;
	ErrorDescription:='Threshold_motorsTargetPosCalculate';
	FB_PlcEmergencyStop();
END_IF
END_ACTION

ACTION A_OneKeyToMaxGap:
//0.上升沿触发
//1.判断电机是否在开启状态,没有就打开电源
//2.判断是否在Moving状态,若有就Stop
//3.将磁间隙打开到至最大阈值
//4.到位后给出反馈
OneKeyToMaxGap_RTRIG(CLK:=btn_OneKeyToMaxGap);
IF OneKeyToMaxGap_RTRIG.Q THEN
	OneKeyToMaxGap_Triggered:=TRUE;
	OneKeyToMaxGap_Done:=FALSE;
END_IF
IF OneKeyToMaxGap_Triggered THEN
	CASE OneKeyToMaxGap_State OF
		0://1.判断电机是否在开启状态,没有就打开电源
			IF st_Power=1 THEN
				OneKeyToMaxGap_State:=1;
			ELSE
				btn_PowerOn:=TRUE;
				IF btn_PowerOn THEN
					A_PowerOn();
				END_IF
			END_IF
		1://1.判断是否在谱学扫描模式，如果是，则切换回正常运动模式
			IF IsSSMotionMode THEN
				SS_Stop:=TRUE;
				IsSSMotionMode:=FALSE;
			END_IF
			OneKeyToMaxGap_State:=2;
		2://判断是否在taper，如果在taper,则判断是否在运动，如果是，则停止运动,0.5sh后，转入下一步
			//IF TaperOrNot THEN
			//	IF moveStatusLeftTop OR moveStatusRightTop OR moveStatusLeftBottom OR moveStatusRightBottom THEN
			//		btn_UserGapStop:=TRUE;
			//	ELSE
			//		OneKeyToMaxGap_TON_Stop2Move_InTaperMode(PT:=T#0.5S);
			//		OneKeyToMaxGap_TON_Stop2Move_InTaperMode.IN:=TRUE;
			//		IF OneKeyToMaxGap_TON_Stop2Move_InTaperMode.Q THEN
			//			TaperOrNot:=FALSE;//关闭taper模式
			//			OneKeyToMaxGap_State:=3;
			//			OneKeyToMaxGap_TON_Stop2Move_InTaperMode.IN:=FALSE;
			//		END_IF
			//	END_IF
			//ELSE
				OneKeyToMaxGap_State:=3;
			//END_IF
		3://3.判断是否在Moving状态,若有就Stop.Taper模式已处理完，此处开始走正常GAP开合逻辑
			IF moveStatusPhaseShifterLin THEN
				btn_UserGapStop:=TRUE;
			ELSE
				OneKeyToMaxGap_TON_Stop2Move(PT:=T#0.5S);
				OneKeyToMaxGap_TON_Stop2Move.IN:=TRUE;
				IF OneKeyToMaxGap_TON_Stop2Move.Q THEN
					OneKeyToMaxGap_State:=4;
					OneKeyToMaxGap_TON_Stop2Move.IN:=FALSE;
				END_IF
			END_IF
		4://4.将磁间隙打开到至最大阈值
			OneKeyToMaxGap_TON(PT:=INT_TO_TIME(LREAL_TO_INT(max_UserGapPositionNew+30))*1000);
			OneKeyToMaxGap_TON.IN:=TRUE;
			OneKeyToMaxGap_TON_Power2Move(PT:=T#0.1S);
			OneKeyToMaxGap_TON_Power2Move.IN:=TRUE;
			UserGapPositionNew:=max_UserGapPositionNew;
			UserGapVelocityNew:=1;
			btn_UserGapMove:=TRUE;
			IF OneKeyToMaxGap_TON_Power2Move.Q THEN
				OneKeyToMaxGap_TON_Power2Move.IN:=FALSE;
				IF FB_MOVE.BCGapDone THEN
					OneKeyToMaxGap_State:=88;
				END_IF
			END_IF
			IF OneKeyToMaxGap_TON.Q THEN//如果150s后，还没有运动到指定gap，则报错
				OneKeyToMaxGap_TON.IN:=FALSE;
				OneKeyToMaxGap_State:=-100;
			END_IF
			IF  btn_UserGapStop THEN
				//
				OneKeyToMaxGap_State:=0;
				OneKeyToMaxGap_Triggered:=FALSE;
				btn_OneKeyToMaxGap:=FALSE;
				OneKeyToMaxGap_Triggered:=FALSE;
				OneKeyToMaxGap_State:=0;
			END_IF
		88://6.到位后给出反馈
			OneKeyToMaxGap_Done:=TRUE;	
			Error:=FALSE;
			ErrorID:=0;
			ErrorDescription:='';
			btn_OneKeyToMaxGap:=FALSE;
			OneKeyToMaxGap_Triggered:=FALSE;
			OneKeyToMaxGap_State:=0;
				
		-100:
			OneKeyToMaxGap_Done:=FALSE;
			Error:=TRUE;
			ErrorID:=1705;
			ErrorDescription:='OneKeyToMaxGap Fail';
			btn_OneKeyToMaxGap:=FALSE;
			OneKeyToMaxGap_Triggered:=FALSE;
			OneKeyToMaxGap_State:=0;
	END_CASE
END_IF
END_ACTION

ACTION A_PowerOff:
CASE d_state OF
		0:(*PowerOff*)
			FB_Power(Off:=TRUE);
				d_state:=1;
		1:
			IF NOT FB_power.OffStatus THEN
				d_state:=1;
			ELSE
				d_state:=88;
			END_IF
		88:(*ResetAllState*)
			btn_PowerOn:=FALSE;
			btn_UserGapMove:=FALSE;
			btn_UserGapStop:=FALSE;
			fb_ton1.IN:=FALSE;
			fb_ton2.IN:=FALSE;
			fb_ton3.IN:=FALSE;
			State:=0;
			Busy:=FALSE;
			InitPowerDone:=FALSE;
			InitCompensationDatasDone:=FALSE;
			Error:=FALSE;
			ErrorID:=0;
			m_state:=0;
			n_state:=0;
			s_state:=0;
			btn_PowerOff:=FALSE;
			d_state:=0;
			Led_Run:=FALSE;
			Led_Error:=FALSE;
			moni_State:=0;
			i:=0;
END_CASE
END_ACTION

ACTION A_PowerOn:
(****************************************************************
NAME:			A_PowerOn
DATA:			2018.1.9
VERSION:		1.0.0
DESCRIPTION:	
				ÉÏµãÃüÁîºó£¬Ë³ÐòÖ´ÐÐ£º
				1.FB_PowerOn
				·µ»ØÖ´ÐÐÊÇ·ñ³É¹¦
HISTORY:
				2019.1.9		NEW

***************************************************************)
fb_ton3(PT:=t#0.5s);
CASE State OF
	0:	(*FB_Power_On*)
		FB_Power(On:=TRUE);
		fb_ton3.IN:=TRUE;
		State:=1;
	1:	(*wait*)
		FB_power();
		IF NOT FB_power.OnStatus THEN		(*FB_Power_OnÃ»ÓÐÖ´ÐÐÍê£¬wait£¬³¬Ê±FB Error*)
			IF NOT fb_ton3.Q THEN
				State:=1;
			ELSE
				ErrorID:=1;
				State:=99;
			END_IF
		ELSE
			State:=88;
		END_IF
	88:	(*All Done*)
		btn_PowerOn:=FALSE;
		State:=0;
		Error:=FALSE;
		ErrorID:=0;
		Busy:=FALSE;
		InitPowerDone:=TRUE;
		FB_power.On:=FALSE;
		fb_ton3.IN:=FALSE;
		LED_Error:=FALSE;
	99:
		Error:=TRUE;
		//ErrorID:=701;
		//ErrorDescription:='power on error';		
		btn_PowerOn:=FALSE;
		State:=99;
		Busy:=FALSE;
		InitPowerDone:=FALSE;
		fb_ton3.IN:=FALSE;
		LED_Error:=TRUE;
END_CASE
END_ACTION

ACTION A_RegularMotion:

(*分别比较四轴目标位置与当前位置的差，如果目标位置比当前位置低，则需要运动到更低-回程差一半；再运动至最终目标位置*)
//只在m=和n=0的时候判断，否则会出现一些BUG，比如往大间隙开时，运动到位后m不能回到0.
IF m_state=0 AND n_state=0 THEN
		TargetPosLessThanCurrentPos:=FALSE;
	IF PhaseShifterLinPositionNew-Pos_PhaseShifterLin<-LEDriftErrorThreshold THEN
			TargetPosLessThanCurrentPos:=TRUE;
	END_IF
END_IF

(*Move*)
IF InitCompensationDatasDone THEN
		(*四轴目标位置都大于当前位置，直接走到目标位置即可，不需要先走到考虑回城误差的临时位置*)
		IF NOT TargetPosLessThanCurrentPos AND NOT HysteresisMoving THEN
			CASE m_state OF
				0:
					FB_Move.Mode:=1;						//1.gap;2.single;3.taper;4.debug;5.BCGap&UserMode		
					FB_Move.PowerState:=st_Power;						
			
					IF btn_UserGapMove THEN				
						moveStatusGap:=TRUE;
						FB_Move.BCGapReset:=TRUE;
						IF NOT st_Power THEN
							ErrorID:=1501;
							Error:=TRUE;
							ErrorDescription:='Plz PowerOn Frist';
							LED_Error:=TRUE;
							//btn_UserGapMove:=FALSE;
							RETURN;
						ELSE
							ErrorID:=0;
							Error:=FALSE;
							ErrorDescription:='';
							LED_Error:=FALSE;
							//btn_UserGapMove:=TRUE;
						END_IF
						//目标速度位置赋值
						FB_Move.TargetGapPosition:=PhaseShifterLinPositionNew;
						FB_Move.TargetGapVelocity:=UserGapVelocityNew;

						m_state:=1;
						FB_Move();
					END_IF
				1:						
					FB_Move.BCGapMove:=TRUE;
					btn_UserGapMove:=FALSE;
					FB_Move();
					IF NOT FB_Move.BCGapDone THEN	
						Led_Run:=TRUE;
						m_state:=1;
					ELSE				
						m_state:=88;
					END_IF
				88:
					moveStatusGap:=FALSE;
					btn_UserGapMove:=FALSE;		
					Led_Run:=FALSE;
					m_state:=0;
			END_CASE
		(*四轴有目标位置小于当前位置，先走到临时位置，再走到目标位置*)
		ELSE
			CASE n_state OF
				0:
					FB_Move.Mode:=1;						//1.gap;2.single;3.taper;4.debug;5.BCGap&UserMode;5:userMode_2		
					FB_Move.PowerState:=st_Power;			
					IF btn_UserGapMove THEN	
						FB_Move.BCGapReset:=TRUE;					
						moveStatusGap:=TRUE;
						IF NOT st_Power THEN
							ErrorID:=1501;
							Error:=TRUE;
							ErrorDescription:='Plz PowerOn Frist';
							LED_Error:=TRUE;
							//btn_UserGapMove:=FALSE;
							RETURN;
						ELSE
							ErrorID:=0;
							Error:=FALSE;
							ErrorDescription:='';
							LED_Error:=FALSE;
							//btn_UserGapMove:=TRUE;
						END_IF						
						//
						IF TargetPosLessThanCurrentPos THEN			
							FB_Move.TargetGapPosition:=PhaseShifterLinPositionNew-HysteresisError;
						ELSE
							FB_Move.TargetGapPosition:=PhaseShifterLinPositionNew;	
						END_IF
						//	
						//	close gap情况下，加入了LeftTopLinPositionNewTemp。//
						//如果在往小间隙运行过程中，改变了目标gap，会在第到达第一次目标位置后，继续向第二
						//次输入的目标运动，而不会回到第一次的目标位置。用temp锁定目标位置
						PhaseShifterLinPositionNewTemp:=PhaseShifterLinPositionNew;
						FB_Move.TargetGapVelocity:=UserGapVelocityNew;
						IF UserGapVelocityNew >1 THEN								  
							ErrorID:=1502;
							Error:=TRUE;
							ErrorDescription:='UserGapVelocityNew must<=1';
							LED_Error:=TRUE;
							btn_UserGapMove:=FALSE;
							RETURN;
						ELSE
							ErrorID:=0;
							Error:=FALSE;
							ErrorDescription:='';
							LED_Error:=FALSE;	
						END_IF										

						FB_Move();
						HysteresisMoving:=TRUE;		
						n_state:=1;	
					END_IF
				1:
					btn_UserGapMove:=FALSE;	
					FB_Move.BCGapMove:=TRUE;
					FB_Move();
					IF NOT FB_Move.BCGapDone THEN			(*还未运动到位置,运动过程中*)
						Led_Run:=TRUE;
						n_state:=1;
					ELSE									
						n_state:=2;							(*转到下一步，运动到最终位置*)
						FB_Move.BCGapMove:=FALSE;
						//Led_Run:=FALSE;
					END_IF
				2:
					FB_Move.BCGapReset:=FALSE;
					FB_Move.Mode:=1;						//1.gap;2.single;3.taper;4.debug;5.BCGap&UserMode		
					FB_Move.PowerState:=st_Power;			
					FB_Move.BCGapMove:=TRUE;
					//直接走到目标位置，已经走到位置的，可以继续下命令，只不过它不在走了而已
					FB_Move.TargetGapPosition:=PhaseShifterLinPositionNewTemp;
					FB_Move.TargetGapVelocity:=UserGapVelocityNew;

					FB_Move();							
					n_state:=3;
				3:
					FB_Move();
					IF NOT FB_Move.BCGapDone THEN			(*还未运动到位置,运动过程中*)
						Led_Run:=TRUE;
						n_state:=3;
					ELSE									
						n_state:=88;							(*运动到了最终位置*)
					END_IF
					(*
					IF NOT Unreach_LS_Bottom THEN
						n_state:=88;							(*在运动过程中如果碰到下限位，则也转到下一步，运动到最终位置*)
						FB_Move.BCGapMove_2:=FALSE;
					END_IF
					*)
				88:				
					moveStatusGap:=FALSE;
					btn_UserGapMove:=FALSE;				
					Led_Run:=FALSE;
					n_state:=0;
					HysteresisMoving:=FALSE;
			END_CASE
		END_IF
	//
	//FB_Move.BCLeftTopPosition等四轴位置监控
	//
END_IF


CASE s_state OF
	0:
		IF btn_UserGapStop OR btn_Reset THEN					
			moveStatusGap:=FALSE;
			m_state:=0;	
			n_state:=0;	
			HysteresisMoving:=FALSE;
			
			FB_Stop.Mode:=1;	
			FB_Stop.PowerState:=st_Power;
			FB_Stop.BCGapStop:=TRUE;
			FB_Stop();	
			s_state:=1;
		END_IF
	1:
		btn_UserGapStop:=FALSE;	
		FB_Stop();
		IF NOT FB_Stop.BCGapDone THEN
			s_state:=1;
		ELSE
			s_state:=88;
		END_IF
	88:
		FB_Move.BCGapReset:=FALSE;
		btn_reset:=FALSE;
		s_state:=0;
END_CASE


(*触发限位开关后，相当于点击了Stop按钮*)
FTrig_ReachLS(CLK:=Unreach_LS_Far AND Unreach_LS_Near);
IF FTrig_ReachLS.Q THEN
	btn_UserGapStop:=TRUE;
END_IF
(*触发限位后，如果继续向前运动，点击move，则相当于点击stop，用于恢复move的状态位*)
IF NOT Unreach_LS_Far AND btn_UserGapMove AND UserGapPositionNew >= UserGapPositionDisplay THEN
	btn_UserGapStop:=TRUE;
END_IF
IF NOT Unreach_LS_Near AND btn_UserGapMove AND UserGapPositionNew <= UserGapPositionDisplay THEN
	btn_UserGapStop:=TRUE;
END_IF
END_ACTION

ACTION A_SpectroscopyScanningMotion:
(*输入保护*)
IF SS_Move AND SSMotionMode AND NOT RegularMotionMode THEN
	IF NOT inRange_SS_StepSize THEN
		SS_Stop:=TRUE;
		SS_Move:=FALSE;
		Error:=TRUE;
		ErrorId:=805;
		ErrorDescription:='target StepSize out of range,please check';
		RETURN;
	ELSE
		//SS_Stop:=FALSE;
		Error:=FALSE;
		ErrorId:=0;
		ErrorDescription:='';	
	END_IF
	//
	IF NOT inRange_SS_StepNumber THEN
		SS_Stop:=TRUE;
		SS_Move:=FALSE;
		Error:=TRUE;
		ErrorId:=806;
		ErrorDescription:='target StepNumber out of range,please check';
		RETURN;
	ELSE
		//SS_Stop:=FALSE;
		Error:=FALSE;
		ErrorId:=0;
		ErrorDescription:='';	
	END_IF
	IF NOT inRange_SS_StepVelocity THEN
		SS_Stop:=TRUE;
		SS_Move:=FALSE;
		Error:=TRUE;
		ErrorId:=807;
		ErrorDescription:='target StepVelocity out of range,please check';
		RETURN;
	ELSE
		//SS_Stop:=FALSE;
		Error:=FALSE;
		ErrorId:=0;
		ErrorDescription:='';	
	END_IF
	IF NOT inRange_StepEachTime_ms THEN
		SS_Stop:=TRUE;
		SS_Move:=FALSE;
		Error:=TRUE;
		ErrorId:=808;
		ErrorDescription:='target StepEachTime_ms out of range,please check';
		RETURN;
	ELSE
		//SS_Stop:=FALSE;
		Error:=FALSE;
		ErrorId:=0;
		ErrorDescription:='';	
	END_IF
END_IF
(*单步时长转换*)
StepEachTime:=INT_TO_TIME(StepEachTime_ms);
SS_TON(PT:=StepEachTime);
(*上升沿触发，初始SS位置=当前磁间隙*)
RTRG_SS_StartPositionDisplay(CLK:=SS_Move);
IF RTRG_SS_StartPositionDisplay.Q THEN
	SS_StartPositionDisplay:=UserGapPositionDisplay;
	SS_InitStartPositionDone:=TRUE;
END_IF
(*SS主程序*)
IF InitPowerDone AND InitCompensationDatasDone AND SS_Move AND SS_InitStartPositionDone THEN
	CASE SS_MoveState OF
		0:
				//UserGapPositionNew:=UserGapPositionDisplay+SS_StepSize;
				UserGapPositionNew:=SS_StartPositionDisplay+SS_StepSize*(SS_currentStep+1);
				A_InitCompensationData();
				FB_Move.Mode:=1;						//1.gap;2.single;3.taper;4.debug;5.BCGap&UserMode		
				FB_Move.PowerState:=st_Power;							
				FB_Move.TargetGapPosition:=PhaseShifterLinPositionNew;
				FB_Move.TargetGapVelocity:=UserGapVelocityNew;		
				FB_Move.BCGapMove:=TRUE;
				FB_Move();
				SS_MoveState:=1;
		1:
				SS_TON.IN:=TRUE;
				FB_Move();
				IF FB_Move.GapMoving AND NOT SS_TimeCountBegin THEN
					SS_StepSystemTime_Begin[SS_currentStep]:=F_GetSysTime();
					SS_TimeCountBegin:=TRUE;
				END_IF
				IF NOT FB_Move.BCGapDone THEN			
					Led_Run:=TRUE;
					SS_MoveState:=1;
				ELSE									
					SS_MoveState:=66;
					SS_StepSystemTime_End[SS_currentStep]:=F_GetSysTime();
					SS_StepCountTime[SS_currentStep]:=SS_StepSystemTime_End[SS_currentStep]-SS_StepSystemTime_Begin[SS_currentStep];
					SS_TimeCountBegin:=FALSE;
				END_IF
		66:
				SS_currentStep:=SS_currentStep+1;			
				Led_Run:=FALSE;
				IF SS_currentStep=SS_StepNumber THEN								
					SS_MoveState:=88;
				END_IF
				IF SS_currentStep<SS_StepNumber THEN
					SS_MoveState:=77;
				END_IF
		77://等待单步时长够
				IF SS_TON.Q THEN
					SS_TON.IN:=FALSE;
					SS_MoveState:=0;
				END_IF
		88:
				SS_TON.IN:=FALSE;
				SS_Move:=FALSE;	
				Led_Run:=FALSE;
				SS_MoveState:=0;
				SS_currentStep:=0;
				SS_InitStartPositionDone:=FALSE;
				//SS_StepSystemTime[SS_StepNumber]:=F_GetSysTime();
	END_CASE
END_IF
(*获取每一步耗时*)
//FOR	m:= 0 TO SS_StepNumber DO
//	SS_StepCountTime[m]:=(SS_StepSystemTime_End[m]-SS_StepSystemTime_Begin[m]);
//END_FOR

(*STOP*)
IF SS_Stop THEN
	FB_Move.BCGapReset:=TRUE;							(*¸øÔË¶¯FB¸øÍ£Ö¹ÐÅºÅ£¬Ê¹FB_Move×´Ì¬»Ö¸´*)
	FB_Move();											(*Æô¶¯FB_Move*)
	SS_Move:=FALSE;								(*btn_GapMove:=FALSE*)
	SS_MoveState:=0;										(*m_state:=0;*)
	CASE SS_StopState OF
			0:
				FB_Stop.Mode:=1;							(*1£ºgapÄ£Ê½£»2£ºµ¥ÁºÄ£Ê½£»3£ºtaperÄ£Ê½£»4£ºDebugÄ£Ê½£»5£ºBCGapÄ£Ê½*)
				FB_Stop.PowerState:=st_Power;				(*µçÔ´×´Ì¬ÊäÈë*)
				FB_Stop.BCGapStop:=TRUE;				(*Execute TRUE*)
				FB_Stop();								(*Æô¶¯FB*)
				SS_StopState:=1;
			1:
				FB_Stop();
				IF NOT FB_Stop.BCGapDone THEN			(*Í£Ö¹Î´Íê³É£¬Ñ­»·*)
					SS_StopState:=1;
				ELSE									(*Í£Ö¹Íê³É£¬ÏÂÒ»²½*)
					SS_StopState:=88;
				END_IF
			88:
				SS_Stop:=FALSE;						(*»Ö¸´×´Ì¬*)
				FB_Move.BCGapReset:=FALSE;				(*ÔËÐÐFB*)
				SS_StopState:=0;
		END_CASE
END_IF

(*触发限位开关后，相当于点击了Stop按钮*)
FTrig_ReachLS(CLK:=Unreach_LS_Far AND Unreach_LS_Near);
IF FTrig_ReachLS.Q THEN
	SS_Stop:=TRUE;
END_IF
END_ACTION

END_PROGRAM

// ---- POUs/CommonFB/MainFB/FB_SetAxisPosition.TcPOU
(****************************************************************
NAME:			FB_SetAxisPosition
DATA:			2017.2.16
VERSION:		1.0.0
DESCRIPTION:	FB_SetAxisPosition
HISTORY:
				2017.2.16		NEW

***************************************************************)
FUNCTION_BLOCK FB_SetAxisPosition
VAR_INPUT
	//GapValueSet:LREAL:=0;
	ValueSet_PhaseShifterLin:LREAL:=0;
	Execute:BOOL;
END_VAR
VAR_OUTPUT
	FbID:DINT:=1001;
	State:DINT;
	Busy:BOOL;
	Done:BOOL;
	Error:BOOL;
	ErrorID:DINT;
END_VAR
VAR
	PhaseShifterLin_MC_SetPosition: MC_SetPosition;
	fb_ton: TON;
	FB_PlcEmergencyStop: FB_PlcEmergencyStop;
END_VAR

IF Execute THEN
Busy:=TRUE;
Done:=FALSE;
fb_ton(PT:=t#0.1s);
CASE State OF
	0:
		IF PhaseShifterLin_MC_SetPosition.Error  THEN		(*FB Error*)
			ErrorID:=1;
			State:=99;
		END_IF
		State:=1;
	1:	(*Execute*)
		PhaseShifterLin_MC_SetPosition.Position:=ValueSet_PhaseShifterLin;
		PhaseShifterLin_MC_SetPosition.Execute:=TRUE;
		A_SetPositionMC();
		fb_ton.IN:=TRUE;
		State:=2;
	2:	(*Wait*)
		A_SetPositionMC();
		IF NOT PhaseShifterLin_MC_SetPosition.Done THEN		(*DoneÐÅºÅ²»µ½£¬¼ÌÐøµÈ´ý£¬Èç¹û³¬Ê±ÔòFB Error*)
			IF NOT fb_ton.Q THEN
				State:=2;
			ELSE
				ErrorID:=4;
				State:=99;
			END_IF
		ELSIF  PhaseShifterLin_MC_SetPosition.Done THEN		(*Done£¬×ªÏÂÒ»²½*)
			State:=88;
		ELSE
			ErrorID:=5;
			State:=99;
		END_IF
	88:
		Execute:=FALSE;
		State:=0;
		Busy:=FALSE;
		Done:=TRUE;
		Error:=FALSE;
		ErrorID:=0;
		PhaseShifterLin_MC_SetPosition.Execute:=FALSE;
		fb_ton.IN:=FALSE;
	99:
		Execute:=FALSE;
		State:=99;
		Busy:=FALSE;
		Done:=FALSE;
		Error:=TRUE;
		PhaseShifterLin_MC_SetPosition.Execute:=FALSE;
		fb_ton.IN:=FALSE;
	-100:
		FB_PlcEmergencyStop();
		Execute:=FALSE;
		State:=-100;
		Busy:=FALSE;
		Done:=FALSE;
		Error:=TRUE;
		PhaseShifterLin_MC_SetPosition.Execute:=FALSE;
		fb_ton.IN:=FALSE;
END_CASE
END_IF

ACTION A_SetPositionMC:
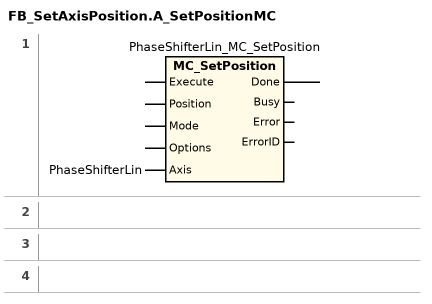
// NETWORK 1
PhaseShifterLin_MC_SetPosition(Axis := PhaseShifterLin); // MC_SetPosition

// NETWORK 2

// NETWORK 3

// NETWORK 4
END_ACTION

END_FUNCTION_BLOCK

// ---- POUs/CommonFB/MainFB/FB_SetMotorAxisPosition.TcPOU
(****************************************************************
NAME:			FB_SetAxisPosition
DATA:			2017.2.16
VERSION:		1.0.0
DESCRIPTION:	FB_SetAxisPosition
HISTORY:
				2017.2.16		NEW

***************************************************************)
FUNCTION_BLOCK FB_SetMotorAxisPosition
VAR_INPUT
	//GapValueSet:LREAL:=0;
	ValueSet_PhaseShifterMotor:LREAL:=0;
	Execute:BOOL;
END_VAR
VAR_OUTPUT
	FbID:DINT:=1001;
	State:DINT;
	Busy:BOOL;
	Done:BOOL;
	Error:BOOL;
	ErrorID:DINT;
END_VAR
VAR
	PhaseShifterMotor_MC_SetPosition: MC_SetPosition;
	fb_ton: TON;
	FB_PlcEmergencyStop: FB_PlcEmergencyStop;
END_VAR

IF Execute THEN
Busy:=TRUE;
Done:=FALSE;
fb_ton(PT:=t#0.1s);
CASE State OF
	0:
		IF PhaseShifterMotor_MC_SetPosition.Error  THEN		(*FB Error*)
			ErrorID:=1;
			State:=99;
		END_IF
		State:=1;
	1:	(*Execute*)
		PhaseShifterMotor_MC_SetPosition.Position:=ValueSet_PhaseShifterMotor;
		PhaseShifterMotor_MC_SetPosition.Execute:=TRUE;
		A_SetMotorPositionMC();
		fb_ton.IN:=TRUE;
		State:=2;
	2:	(*Wait*)
		A_SetMotorPositionMC();
		IF NOT PhaseShifterMotor_MC_SetPosition.Done THEN		(*DoneÐÅºÅ²»µ½£¬¼ÌÐøµÈ´ý£¬Èç¹û³¬Ê±ÔòFB Error*)
			IF NOT fb_ton.Q THEN
				State:=2;
			ELSE
				ErrorID:=4;
				State:=99;
			END_IF
		ELSIF  PhaseShifterMotor_MC_SetPosition.Done THEN		(*Done£¬×ªÏÂÒ»²½*)
			State:=88;
		ELSE
			ErrorID:=5;
			State:=99;
		END_IF
	88:
		Execute:=FALSE;
		State:=0;
		Busy:=FALSE;
		Done:=TRUE;
		Error:=FALSE;
		ErrorID:=0;
		PhaseShifterMotor_MC_SetPosition.Execute:=FALSE;
		fb_ton.IN:=FALSE;
	99:
		Execute:=FALSE;
		State:=99;
		Busy:=FALSE;
		Done:=FALSE;
		Error:=TRUE;
		PhaseShifterMotor_MC_SetPosition.Execute:=FALSE;
		fb_ton.IN:=FALSE;
	-100:
		FB_PlcEmergencyStop();
		Execute:=FALSE;
		State:=-100;
		Busy:=FALSE;
		Done:=FALSE;
		Error:=TRUE;
		PhaseShifterMotor_MC_SetPosition.Execute:=FALSE;
		fb_ton.IN:=FALSE;
END_CASE
END_IF

ACTION A_SetMotorPositionMC:
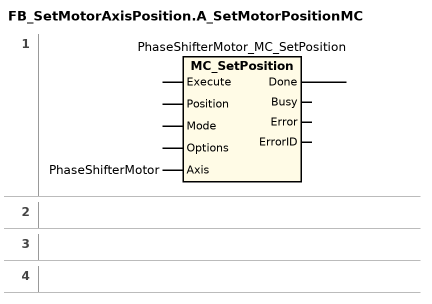
// NETWORK 1
PhaseShifterMotor_MC_SetPosition(Axis := PhaseShifterMotor); // MC_SetPosition

// NETWORK 2

// NETWORK 3

// NETWORK 4
END_ACTION

END_FUNCTION_BLOCK

// ---- POUs/MAIN.TcPOU
PROGRAM MAIN
VAR
	fb_led_Show: FB_LedShow;
	btn_reset: BOOL;
	CPMU_PLC_Reset: PLC_Reset;
	d_state: DINT;
	CPMU_PLC_Start: PLC_Start;
	powerStatus:BOOL;

(*TwinSAFE*)
	Safe_run AT%Q*:BOOL;
	Err_Ack AT %Q*:BOOL;
	Estop_RunAndRestart AT %Q*:BOOL;
	AX5805_Error_Ack AT %Q*:BOOL;
	Led_Run  AT %Q*:BOOL;
	Led_Error  AT %Q*:BOOL;

	FB_ERROR AT%I*:BOOL;
	COM_ERROR AT%I*:BOOL;
	//OUT_ERROR AT%I*:BOOL;
	Estop_Out AT%I*:BOOL;

	SafeStatus:INT;
	SafePLCRunOK: BOOL;
	fb_ton: TON;
	fb_ton2: TON;
	fb_ton3: TON;
	fb_ton1: TON;
	fb_ton0: TON;
(*IO*)
	el1808_D1  AT%I* :ARRAY[1..4] OF BOOL;
	el1008 AT%I*:BOOL;
	EStopTrig:BOOL;
(*setAxisPosition*)
	SetAxisPosState: INT;
	FB_Set_AxisPosition:FB_SetAxisPosition;
	fb_ton4: TON;
	fb_ton5: TON;
	fb_ton6: TON;
	SetAxisPositionDone: BOOL;

	i: INT;
	j: INT;

(****RS232***)
	fbEL6001	: FB_SerialCom;
	
	moveDonePhaseShifter: BOOL;


(*Torque*)
	Torque_PS AT%I*:INT;
(**)
	btn_setAxisPosition: BOOL;
	ValueSet_PhaseShifterLin:LREAL;
(**)
	RestartTC: TC_Restart;
	
(*recipe*)
	RecipeINT:INT;
	RecipeBOOL:BOOL;
	RecipeManCommands: RecipeManCommands;
	SaveParameter : BOOL;  //保存文件
	LoadParameter : BOOL;  //读取文件
	Save_R_TRIG   : R_TRIG;
	Read_R_TRIG   : R_TRIG;
	loadparameterStatus: INT;
	RecipeBOOL2:BOOL;
	ReturnDwordLoad: DWORD;
	InsertionDeviceName:STRING;
(*UserMode*)
	pbUserMode: BOOL:=TRUE;
	EL1904 AT%I* :ARRAY[1..24] OF BOOL;
	setAxisPositionEnable: BOOL;
	state_loadParameters: INT;
	state_setLEPosBias: INT;
	//
	PositionBiasSet:BOOL;
	MC_SetLEPosBias_PhaseShifter:MC_WriteParameter;
	PositionBias_PhaseShifter: LREAL:=10.1;
	LoadLEPB_R_TRIG: R_TRIG;
	PositionBiasTON: TON;
	
	//
	OPC_TEST_Bi:BOOL:=TRUE; (*~ (OPC:1:available for OPC Clients) *)
	OPC_TEST_Bi2:BOOL;(*~ (OPC:1:available for OPC Clients) *)
	//
	HasTemperatureSensorOrNot:BOOL;//Only IVU or CPMU
	(*Sensor Reading*)
	Sensor_Reading_1 AT %I*:ARRAY[0..3] OF BYTE;
	Sensor_Reading_2 AT %I*:ARRAY[0..3] OF BYTE;
	Sensor_Reading_3 AT %I*:ARRAY[0..3] OF BYTE;
	Sensor_Reading_4 AT %I*:ARRAY[0..3] OF BYTE;
	Sensor_Reading_5 AT %I*:ARRAY[0..3] OF BYTE;
	Sensor_Reading_6 AT %I*:ARRAY[0..3] OF BYTE;
	Sensor_Reading_7 AT %I*:ARRAY[0..3] OF BYTE;
	Sensor_Reading_8 AT %I*:ARRAY[0..3] OF BYTE;
	Sensor_Reading_DpState AT %I*:USINT;
	Sensor_Reading_ExtDiagFlag AT %I*:BOOL;
	TemperatureSensors_1:LREAL;
	TemperatureSensors_2:LREAL;
	TemperatureSensors_3:LREAL;
	TemperatureSensors_4:LREAL;
	TemperatureSensors_5:LREAL;
	TemperatureSensors_6:LREAL;
	TemperatureSensors_7:LREAL;
	TemperatureSensors_8:LREAL;
	dut_sensor_datas_1:DUT_SENSOR_DATAS_1;
	dut_sensor_datas_2:DUT_SENSOR_DATAS_2;
	dut_sensor_datas_3:DUT_SENSOR_DATAS_3;
	dut_sensor_datas_4:DUT_SENSOR_DATAS_4;
	dut_sensor_datas_5:DUT_SENSOR_DATAS_5;
	dut_sensor_datas_6:DUT_SENSOR_DATAS_6;
	dut_sensor_datas_7:DUT_SENSOR_DATAS_7;
	dut_sensor_datas_8:DUT_SENSOR_DATAS_8;
	//
	temperature_gradient_2_To_1:LREAL;
	temperature_gradient_3_To_2:LREAL;
	temperature_gradient_5_To_4:LREAL;
	temperature_gradient_6_To_5:LREAL;
	temperature_gradient_max:LREAL;
	//
	temperature_average:LREAL;
	A_SetLinearEncoderPositionBias_Enable: BOOL;
	
		//
	temperatureStatus:INT;//0：有传感器度数错误；1:常温；2:低温；3:常温和低温中间态
	CryogenicTemperatureThreshold:LREAL:=80;//80K以下归划分为低温
	RoomTemperatureThreshold:LREAL:=293;//293K以上划分为常温
	//CPMU cryogenix ON/FF
	CryogenicCompensationOn:BOOL;
	CryogenicCompensationConditionsReady:BOOL;
	CryogenicCompensation_LeftTop:LREAL;
	CryogenicCompensation_RightTop:LREAL;
	CryogenicCompensation_LeftBottom:LREAL;
	CryogenicCompensation_RightBottom:LREAL;
	CryogenicCompensationDone: BOOL;
	
(**)
	bDriveDiagMessageAndNumber  : BOOL;
	m_GetDriveStatusState:INT;
	GetDriveStatusStateDone:BOOL;
	GetDriveStatusStateError:BOOL;
	GetDriveStatusTON: TON;
	//	
	fb_SoEReadDiagMessage_PhaseShifter: FB_SoEReadDiagMessage;
	DriveDiagMessage_PhaseShifter:STRING;
	//
	FB_SoEReadDiagNumber_PhaseShifter: FB_SoEReadDiagNumber;
	DriveDiagNumber_PhaseShifter:UDINT;
	bReloadDriveDiagMessageAndNumber: BOOL;
	
	(*load IOC*)
	bExe_load_Prog: BOOL;
	NT_StartProcess_Load: NT_StartProcess;
	Exe_load_step: UINT;
	R_TRIG_ExeLoad: R_TRIG;
	Exe_Load_Done:BOOL;
	(*kill IOC*)
	bExe_Kill_Prog: BOOL;
	NT_StartProcess_Kill: NT_StartProcess;
	Exe_kill_step: UINT;
	R_TRIG_Exekill: R_TRIG;
	Exe_Kill_Done:BOOL;

	KS_RightBottom_Near_Contact2: BOOL;
	
	//
	//more parameters get:gear;feedback2 direction 
	//
	//GetMoreDriveStatus_FunctionON:BOOL:=TRUE;
	GetDriveStatusTON2: TON;
	//GearNumerator,st182
	st_p182_PhaseShifter:ST_P182;
	FB_SoERead_GearNumerator_PhaseShifter: FB_SoERead;
	GearNumeratorGet_PhaseShifter:UDINT;
	GearNumeratorConfigured_PhaseShifter:UDINT;
	//GearDenominator,st183
	st_p183_PhaseShifter:ST_P183;
	FB_SoERead_GearDenominator_PhaseShifter: FB_SoERead;
	GearDenominatorGet_PhaseShifter:UDINT;
	GearDenominatorConfigured_PhaseShifter:UDINT;
	//Feedback2direction,st180
	st_p180_PhaseShifter:ST_P180;
	FB_SoERead_Feedback2direction_PhaseShifter: FB_SoERead;
	Feedback2directionGet_PhaseShifter:UINT;
	Feedback2directionConfigured_PhaseShifter:UINT;
	//
	//RestartDrivers
		(*重启驱动器*)
	btn_RestartDriversAll:BOOL;
	btn_RestartDriver1:BOOL;
	btn_RestartDriver2:BOOL;
	btn_RestartDriver3:BOOL;
	btn_RestartDriver4:BOOL;
	btn_RestartDriver5:BOOL;
	btn_RestartDriver6:BOOL;
	btn_RestartDriver7:BOOL;
	btn_RestartDriver8:BOOL;
	Relay_EL2624 AT %Q*:ARRAY[0..7]OF  BOOL;
	RestartDriver_RTRIG:R_TRIG;
	RestartDriver_TON:TON;
	RestartDriver_Triggered:BOOL;
	RestartDriver_State:DINT;
	RestartDriver_Done:BOOL;
	
	//
	//	LEHeartBeatMonitorFunction
	//
	LEHeartBeatMonitorFunctionOn: BOOL;
	LEHeartBeatFirstScan:BOOL;
	LEHeartBeatDeadZone : LREAL := 0; 
	LEHeartBeatAlarmTime : TIME := T#0.1S;
	
    //Pos_LeftTopLin_Last : LREAL; 
	Velo_PhaseShifterLin_Last : LREAL; 
	Pos_PhaseShifterMotor_Initial : LREAL; 
    StableTimer_PhaseShifterLin : TON; 
    StableTime_PhaseShifterLin : TIME; 
    DeltaVelo_PhaseShifterLin : LREAL; 
	IsInitialPositionSet_PhaseShifter: BOOL;
	MotorPosChange_PhaseShifter: LREAL;
	Threshold_PhaseShifterMotorPos:LREAL:=0.1;
	Threshold_PhaseShifterMotorVelo:LREAL:=0.2;
	Alarm_PhaseShifterLin:BOOL;
	Alarm_PhaseShifterMotorPos:BOOL;
	Alarm_PhaseShifterMotorVelo:BOOL;
	
	(*setAxisPosition*)
	SetMotorAxisPosState: INT;
	FB_Set_MotorAxisPosition:FB_SetMotorAxisPosition;
	fb_ton4_2: TON;
	fb_ton5_2: TON;
	fb_ton6_2: TON;
	SetMotorAxisPositionDone: BOOL;
	
	btn_SetMotorAxisPosition: BOOL;
	MonitorMotorAndLEFunctionOn:BOOL:=TRUE;
END_VAR

(*加载Ricipe参数*)
A_InitRecipeParameters();
(*Restart TwinCAT*)
IF Global_Variables.m_restartTC THEN
(*首先关闭opcIocShell.exe*)	
	bExe_Kill_Prog:=TRUE;
	A_KillOpcIocShellExe();
(*重启TC*)
	IF Exe_Kill_Done THEN
		A_RestartTC();
	END_IF
END_IF
(*******InitAxisParameters*******)
A_InitAxisParameters();
(*******CheckLimitSwitch*******)
A_CheckLimitSwitch();
(*Check Kill Switch*)
A_CheckKillSwitch();
(*******PosDiff¼à¿Ø*******)
A_PosDiffDetectiion();
(*******³õÊ¼»¯SafePlc*******)
IF NOT simulation THEN
A_SafePlcStartInit();
END_IF
(************SetAxisPosition*********************)
IF  NOT USELinearEncoder AND setAxisPositionEnable AND btn_setAxisPosition THEN
	//IF NOT SerAxisPositionDone THEN
		FB_Set_AxisPosition.ValueSet_PhaseShifterLin:=ValueSet_PhaseShifterLin;
		A_SetAxisPosition();
	//END_IF
END_IF
(*******³Mode Select******)
IF SafePLCRunOK OR Simulation THEN
	UserMode();
END_IF
(*******Led Show******)
fb_led_Show();
(*******Check Power status******)
FB_Power(Check:=TRUE);
st_Power:=FB_Power.PowerState;
(*********RS232*********************)
BackgroundEL();
(*fbEL6001(TxBuffer:=TxBufferEL, RxBuffer:=RxBufferEL);*)

(*设置position bias*)
IF loadParametersDone AND (DriveStatus=1 OR simulation) THEN 
	A_SetLinearEncoderPositionBias();
END_IF
(*检查硬急停状态，包括安全限位、柜门急停、手持急停*)
A_CheckHardwareEmergencyStopStatus();
(*获取驱动器状态信息*)
IF NOT simulation THEN
	A_GetDriverStatus();
END_IF
(*IDControlReady*)
IF ((DriveStatus<>0 AND SafePLCRunOK) OR simulation) AND NOT Error THEN
	IDControlReady:=TRUE;
ELSE
	IDControlReady:=FALSE;
END_IF

(*IOC Start*)
//IF IDControlReady THEN
	bExe_load_Prog:=TRUE;
	A_LoadOpcIocShellExe();
//END_IF

(*检查光栅读数是否在范围内*)
A_CheckLinearEncoder();

(*RestartDrivers*)
A_RestartDrivers();

(*A_LEHeartBeatMonitor*)
IF LEHeartBeatMonitorFunctionOn THEN
	A_LEHeartBeatMonitor();
END_IF
(************SetMotorAxisPosition*********************)
//IDControl 1s after
fb_ton5_2.IN:=IDControlReady;
fb_ton5_2.PT:=T#1S;
fb_ton5_2();
IF fb_ton5_2.Q THEN
	btn_SetMotorAxisPosition:=TRUE;
END_IF
IF  USELinearEncoder AND btn_SetMotorAxisPosition THEN
	IF NOT SetMotorAxisPositionDone THEN
		FB_Set_MotorAxisPosition.ValueSet_PhaseShifterMotor:=Pos_PhaseShifterLin;
		A_SetMotorAxisPosition();
	END_IF
END_IF
(*A_MonitorMotorAndLE*)
IF MonitorMotorAndLEFunctionOn AND SetMotorAxisPositionDone THEN
	A_MonitorMotorAndLE();
END_IF
(*A_CheckMaxVelocity*)
A_CheckMaxVelocity();

ACTION A_CheckHardwareEmergencyStopStatus:
IF 	NOT KS_TopNear_Contact1 OR
	NOT KS_TopNear_Contact2 OR
	NOT KS_TopFar_Contact1 OR
	NOT KS_TopFar_Contact2 OR
	
(*E-STOP*)
	NOT KS_CabinetEmergency_contact1 OR
	NOT KS_CabinetEmergency_contact2 OR
	NOT KS_handEmergency1_Contact1 OR
	NOT KS_handEmergency1_Contact2 OR
	NOT KS_handEmergency2_Contact1 OR
	NOT KS_handEmergency2_Contact2 OR
	NOT KS_softEmergency2_Contact THEN
	Hardware_EmergencyStop:=FALSE;
ELSE
	Hardware_EmergencyStop:=TRUE;
END_IF
END_ACTION

ACTION A_CheckKillSwitch:
IF simulation THEN	
	KS_TopFar_Contact1:=TRUE;	
	KS_TopFar_Contact2:=TRUE;	
	KS_TopNear_Contact1:=TRUE;	
	KS_TopNear_Contact2:=TRUE;	
	KS_BottomFar_Contact1:=TRUE;	
	KS_BottomFar_Contact2:=TRUE;	
	KS_BottomNear_Contact1:=TRUE;	
	KS_BottomNear_Contact2:=TRUE;	
	(*E-STOP*)
	KS_CabinetEmergency_contact1:=TRUE;
	KS_CabinetEmergency_contact2:=TRUE;	
	KS_handEmergency1_Contact1:=TRUE;
	KS_handEmergency1_Contact2:=TRUE;
	KS_handEmergency2_Contact1:=TRUE;
	KS_handEmergency2_Contact2:=TRUE;
	
	KS_softEmergency2_Contact:=TRUE;

ELSE
	KS_TopFar_Contact1:=EL1904[1];//c1	
	KS_TopFar_Contact2:=EL1904[2];//c1	
	KS_TopNear_Contact1:=EL1904[3];//c1	
	KS_TopNear_Contact2:=EL1904[4];//c1	
	KS_BottomFar_Contact1:=EL1904[5];//c2	
	KS_BottomFar_Contact2:=EL1904[6];//c2	
	KS_BottomNear_Contact1:=EL1904[7];//c2	
	KS_BottomNear_Contact2:=EL1904[8];//c2
	
	
	(*E-STOP*)
	KS_CabinetEmergency_contact1:=EL1904[9];//c3
	KS_CabinetEmergency_contact2:=EL1904[10];//c3
	
	KS_handEmergency1_Contact1:=EL1904[11];//c3
	KS_handEmergency1_Contact2:=EL1904[12];//c3
	KS_handEmergency2_Contact1:=EL1904[13];//c4
	KS_handEmergency2_Contact2:=EL1904[14];//c4
	
	KS_softEmergency2_Contact:=EL1904[15];//c4
	//c4
	END_IF
END_ACTION

ACTION A_CheckLimitSwitch:
(*******1.´ÓIO»ñÈ¡ÏÞÎ»×´Ì¬******)
(**)
IF simulation THEN
	(**)
	LS_TopFar  :=TRUE;
	LS_TopNear :=TRUE;
	LS_BottomFar :=TRUE;
	LS_BottomNear  :=TRUE;
ELSE
	LS_TopFar  :=el1808_D1[1];
	LS_TopNear :=el1808_D1[2];
	LS_BottomFar :=el1808_D1[3];
	LS_BottomNear :=el1808_D1[4];

END_IF
(******2.TopÏÞÎ»»òÕßBottomÏÞÎ»ÓÐÒ»¸ö´¥·¢£¬È«¾Ö±äÁ¿¡£¸øMC_POWERÓÃÓÚ·½Ïò¿ØÖÆ£¬ÓÐÒ»¸öÏÞÎ»Îª´¥·¢ÎªFALSE£¬ÔòUnreach_LSÎªFALSE******)
//Unreach_LS_Far:=LS_TopFar AND LS_BottomFar;
//Unreach_LS_Near:=LS_TopNear AND LS_BottomNear;

Unreach_LS_Far:=LS_TopFar;
Unreach_LS_Near:=LS_TopNear;
END_ACTION

ACTION A_CheckLinearEncoder:
//LEProtectionPosition
min_UserLEProtectionGapPosition:=min_UserGapPositionNew-min_ThresholdGapSoft2LEProtection;//回程误差有0.1mm
max_UserLEProtectionGapPosition:=max_UserGapPositionNew+max_ThresholdGapSoft2LEProtection;

//如果没有使用光栅、或者光栅参数没设置好，则不检查光栅位置
IF NOT USELinearEncoder OR NOT PositionBiasDone THEN
	RETURN;
END_IF
IF Pos_PhaseShifterLin <=0 THEN
	ErrorID:=1101;
	Error:=TRUE;
	ErrorDescription:='Pos_PhaseShifterLin <=0';
	FB_PlcEmergencyStop();
	LED_Error:=TRUE;
END_IF
//

IF Pos_PhaseShifterLin >max_UserLEProtectionGapPosition THEN
	ErrorID:=1105;
	Error:=TRUE;
	ErrorDescription:='Pos_PhaseShifterLin >max_UserLEProtectionGapPosition';
	FB_PlcEmergencyStop();
	LED_Error:=TRUE;
END_IF

//
IF Pos_PhaseShifterLin <min_UserLEProtectionGapPosition THEN
	ErrorID:=1109;
	Error:=TRUE;
	ErrorDescription:='Pos_PhaseShifterLin <min_UserLEProtectionGapPosition';
	FB_PlcEmergencyStop();
	LED_Error:=TRUE;
END_IF
END_ACTION

ACTION A_CheckMaxVelocity:
IF NOT USELinearEncoder OR NOT PositionBiasDone OR NOT IDControlReady THEN
	RETURN;
END_IF
IF NOT st_Power THEN
	RETURN;
END_IF
//Monitoring Motor and LE Position/Velocity
MaxVelocityGlobalVelocity:=MAX(max_UserGapVelocityNew,max_UserTaperVelocityNew,UserMode.max_SS_StepVelocity,
			UserMode.Global_ChainProtection_MPS_MoveVelocity,UserMode.Global_ChainProtection_EPS_MoveVelocity);
IF 	ABS(Velo_PhaseShifterLin) > MaxVelocityGlobalVelocity*1.1/2 THEN
	ErrorID:=7001;
	Error:=TRUE;
	ErrorDescription:='ABS(Velo_PhaseShifterLin) > MaxVelocityGlobalVelocity*1.1/2';
	FB_PlcEmergencyStop();
	LED_Error:=TRUE;
END_IF
IF 	ABS(Velo_PhaseShifterMotor) > MaxVelocityGlobalVelocity*1.1/2 THEN
	ErrorID:=7002;
	Error:=TRUE;
	ErrorDescription:='ABS(Velo_PhaseShifterMotor) > MaxVelocityGlobalVelocity*1.1/2';
	FB_PlcEmergencyStop();
	LED_Error:=TRUE;
END_IF
END_ACTION

ACTION A_GetDriverStatus:
//
//DriveMessage/Drive Number/Gear number/feedback2 direction
//
IF bReloadDriveDiagMessageAndNumber THEN
	m_GetDriveStatusState:=0;
	bReloadDriveDiagMessageAndNumber:=FALSE;
END_IF
GetDriveStatusTON(PT:=T#1S);
GetDriveStatusTON2(PT:=T#0.1S);
A_GetDriverStatusMC();
CASE m_GetDriveStatusState OF
	0:
		GetDriveStatusTON.IN:=TRUE;
		m_GetDriveStatusState:=1;
	1:
		IF GetDriveStatusTON.Q THEN
			bDriveDiagMessageAndNumber:=TRUE;
			m_GetDriveStatusState:=2;
		END_IF
	2:
		GetDriveStatusTON.IN:=FALSE;
		DriveDiagMessage_PhaseShifter:=fb_SoEReadDiagMessage_PhaseShifter.sDiagMessage.strData;
		//
		DriveDiagNumber_PhaseShifter:=FB_SoEReadDiagNumber_PhaseShifter.iDiagNumber;
		//
		GearNumeratorGet_PhaseShifter:=st_p182_PhaseShifter.Feedback_2_geat_numerator;
		//
		GearDenominatorGet_PhaseShifter:=st_p183_PhaseShifter.Feedback_2_geat_denominator;
		//
		Feedback2directionGet_PhaseShifter:=st_p180_PhaseShifter.Feedback_direction;
		//
		IF 	NOT fb_SoEReadDiagMessage_PhaseShifter.bBusy
			AND NOT FB_SoEReadDiagNumber_PhaseShifter.bBusy
			AND NOT FB_SoERead_GearNumerator_PhaseShifter.bBusy 
			AND NOT FB_SoERead_GearDenominator_PhaseShifter.bBusy 
			AND NOT FB_SoERead_Feedback2direction_PhaseShifter.bBusy  THEN
				GetDriveStatusTON2.IN:=TRUE;
				IF GetDriveStatusTON2.Q THEN
					m_GetDriveStatusState:=88;
				END_IF
		END_IF
		IF 	fb_SoEReadDiagMessage_PhaseShifter.bError
			OR FB_SoEReadDiagNumber_PhaseShifter.bError
			OR FB_SoERead_GearNumerator_PhaseShifter.bError 
			OR FB_SoERead_GearDenominator_PhaseShifter.bError 
			OR FB_SoERead_Feedback2direction_PhaseShifter.bError 
		THEN
			m_GetDriveStatusState:=-100;
		END_IF
		
	88:
		bDriveDiagMessageAndNumber:=FALSE;
		A_GetDriverStatusMC();
		GetDriveStatusStateDone:=TRUE;
		GetDriveStatusStateError:=FALSE;
		//
		(*Drive Status*)
		//D012, Axis state machine: Control and power section ready,53266
		IF DriveDiagNumber_PhaseShifter=16#D012  THEN
			DriveStatus:=1;
		//D013, Axis state machine: Axis in operation,53267
		ELSIF DriveDiagNumber_PhaseShifter=16#D013  THEN
			DriveStatus:=2;
		//D014，Axis state machine: Axis halt.53266和53267中间会经历这么一个状态，算正常状态
		ELSIF DriveDiagNumber_PhaseShifter=16#D014  THEN
			DriveStatus:=3;
		ELSE
			DriveStatus:=0;
		END_IF
		//
		//
		//	//check statusGet and status configured
		IF 	GearNumeratorGet_PhaseShifter<>GearNumeratorConfigured_PhaseShifter 
			OR GearDenominatorGet_PhaseShifter<>GearDenominatorConfigured_PhaseShifter   THEN
				bDriveDiagMessageAndNumber:=FALSE;
				A_GetDriverStatusMC();
				GetDriveStatusStateDone:=FALSE;
				GetDriveStatusStateError:=TRUE;
				Error:=TRUE;
				ErrorId:=1302;
				ErrorDescription:='gearParameters Error';
				Plc_EmergencyStop:=FALSE;
		END_IF
		IF USELinearEncoder THEN
			IF  Feedback2directionGet_PhaseShifter<>Feedback2directionConfigured_PhaseShifter THEN
					bDriveDiagMessageAndNumber:=FALSE;
					A_GetDriverStatusMC();
					GetDriveStatusStateDone:=FALSE;
					GetDriveStatusStateError:=TRUE;
					Error:=TRUE;
					ErrorId:=1303;
					ErrorDescription:='fb2direction Error';
					Plc_EmergencyStop:=FALSE;
			END_IF
		END_IF
		m_GetDriveStatusState:=0;
	-100:
		bDriveDiagMessageAndNumber:=FALSE;
		A_GetDriverStatusMC();
		GetDriveStatusStateDone:=FALSE;
		GetDriveStatusStateError:=TRUE;
		Error:=TRUE;
		ErrorId:=1301;
		ErrorDescription:='GetDriveStatusStateError';
END_CASE
END_ACTION

ACTION A_GetDriverStatusMC:
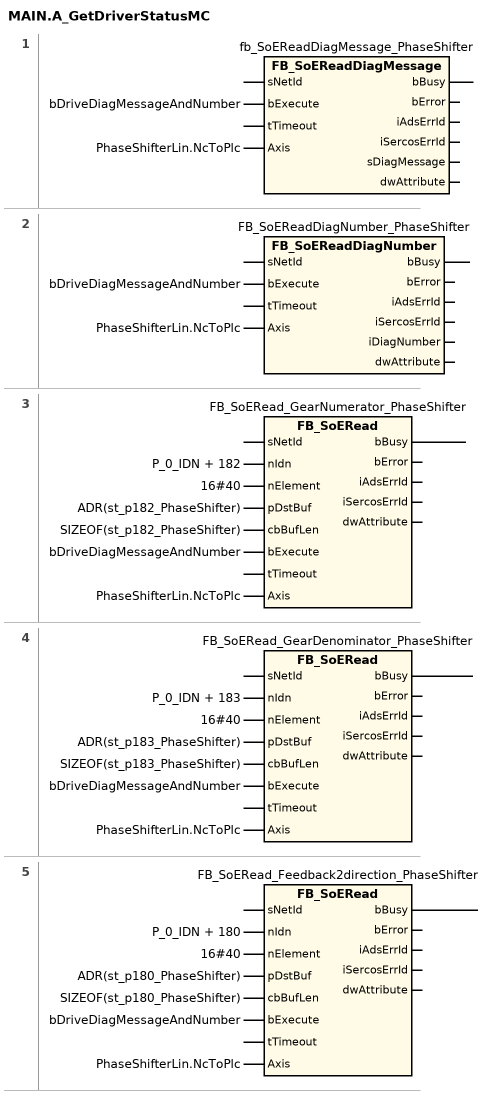
// NETWORK 1
fb_SoEReadDiagMessage_PhaseShifter(bExecute := bDriveDiagMessageAndNumber, Axis := PhaseShifterLin.NcToPlc); // FB_SoEReadDiagMessage

// NETWORK 2
FB_SoEReadDiagNumber_PhaseShifter(bExecute := bDriveDiagMessageAndNumber, Axis := PhaseShifterLin.NcToPlc); // FB_SoEReadDiagNumber

// NETWORK 3
FB_SoERead_GearNumerator_PhaseShifter(
    nIdn := P_0_IDN + 182,
    nElement := 16#40,
    pDstBuf := ADR(st_p182_PhaseShifter),
    cbBufLen := SIZEOF(st_p182_PhaseShifter),
    bExecute := bDriveDiagMessageAndNumber,
    Axis := PhaseShifterLin.NcToPlc); // FB_SoERead

// NETWORK 4
FB_SoERead_GearDenominator_PhaseShifter(
    nIdn := P_0_IDN + 183,
    nElement := 16#40,
    pDstBuf := ADR(st_p183_PhaseShifter),
    cbBufLen := SIZEOF(st_p183_PhaseShifter),
    bExecute := bDriveDiagMessageAndNumber,
    Axis := PhaseShifterLin.NcToPlc); // FB_SoERead

// NETWORK 5
FB_SoERead_Feedback2direction_PhaseShifter(
    nIdn := P_0_IDN + 180,
    nElement := 16#40,
    pDstBuf := ADR(st_p180_PhaseShifter),
    cbBufLen := SIZEOF(st_p180_PhaseShifter),
    bExecute := bDriveDiagMessageAndNumber,
    Axis := PhaseShifterLin.NcToPlc); // FB_SoERead
END_ACTION

ACTION A_InitAxisParameters:
//LE	
	Pos_PhaseShifterLin:=DINT_TO_LREAL(LREAL_TO_DINT(PhaseShifterLin.NcToPlc.ActPos*100000))/100000;
	moveStatusPhaseShifterLin:=PhaseShifterLin.Status.Moving;
	Velo_PhaseShifterLin:=DINT_TO_LREAL(LREAL_TO_DINT(PhaseShifterLin.NcToPlc.ActVelo*100000))/100000;
	PosDiff_PhaseShifterLin_actual:=DINT_TO_LREAL(LREAL_TO_DINT(PhaseShifterLin.NcToPlc.PosDiff*100000))/100000;
	Torque_PhaseShifterLin:=PhaseShifterLin.NcToPlc.ActTorque;	
	PhaseShifterLin.ReadStatus();

//Motor
	Pos_PhaseShifterMotor:=DINT_TO_LREAL(LREAL_TO_DINT(PhaseShifterMotor.NcToPlc.ActPos*100000))/100000;
	moveStatusPhaseShifterMotor:=PhaseShifterMotor.Status.Moving;
	Velo_PhaseShifterMotor:=DINT_TO_LREAL(LREAL_TO_DINT(PhaseShifterMotor.NcToPlc.ActVelo*100000))/100000;
	PosDiff_PhaseShifterMotor_actual:=DINT_TO_LREAL(LREAL_TO_DINT(PhaseShifterMotor.NcToPlc.PosDiff*100000))/100000;
	Torque_PhaseShifterMotor:=PhaseShifterMotor.NcToPlc.ActTorque;	
	PhaseShifterMotor.ReadStatus();

//
	//get Delta
	//
	//Delta Pos
	DeltaPos_PhaseShifter:=Pos_PhaseShifterLin - Pos_PhaseShifterMotor;
	//Delta Velocity	
	DeltaVelo_PhaseShifter:=Velo_PhaseShifterLin - Velo_PhaseShifterMotor;
	//Delta lagDistance
	DeltaPosDiff_PhaseShifter_actual:=PosDiff_PhaseShifterLin_actual - PosDiff_PhaseShifterMotor_actual;
	//Delta Torque
	DeltaTorque_PhaseShifter:=Torque_PhaseShifterLin - Torque_PhaseShifterMotor;
END_ACTION

ACTION A_InitRecipeParameters:
CASE state_loadParameters OF
	0:
		LoadParameter:=TRUE;
		Read_R_TRIG(CLK:=LoadParameter , Q=> );
		IF Read_R_TRIG.Q THEN
			state_loadParameters:=1;
		END_IF
	1:
		 ReturnDwordLoad:=RecipeManCommands.LoadAndWriteRecipe(RecipeDefinitionName:='Recipes' , RecipeName:='ParametersPS');
    	 LoadParameter:=FALSE;
		 IF ReturnDwordLoad<>0 THEN
		 	state_loadParameters:=-100;
		ELSE
			LoadRecipeParameters:=TRUE;
			LoadParameter:=FALSE;
			state_loadParameters:=88;
	 	END_IF
	88:
		loadParametersDone:=TRUE;
	-100:
		loadParametersDone:=FALSE;
		Error:=TRUE;
		ErrorId:=101;
		ErrorDescription:='LoadRecipeParameters Error';
		Plc_EmergencyStop:=FALSE;
END_CASE
//Save_R_TRIG(CLK:=SaveParameter , Q=> );
Read_R_TRIG(CLK:=LoadParameter , Q=> );
//IF Save_R_TRIG.Q THEN  //将plc数据以文件形式保存在工控机中
//	 RecipeManCommands.CreateRecipe(RecipeDefinitionName:='Recipes' , RecipeName:='ParametersPS2' );
//	 RecipeManCommands.ReadAndSaveRecipe(RecipeDefinitionName:='Recipes' , RecipeName:='ParametersPS2' );
//	 SaveParameter:=FALSE;
//END_IF
IF Read_R_TRIG.Q THEN  //将工控机中的文件数据读取到plc中
     ReturnDwordLoad:=RecipeManCommands.LoadAndWriteRecipe(RecipeDefinitionName:='Recipes' , RecipeName:='ParametersPS');
     LoadParameter:=FALSE;
	 IF ReturnDwordLoad<>0 THEN
		 Error:=TRUE;
		 ErrorId:=101;
		 ErrorDescription:='LoadRecipeParameters Error';
		 Plc_EmergencyStop:=FALSE;
	 END_IF
END_IF
END_ACTION

ACTION A_KillOpcIocShellExe:
R_TRIG_Exekill(CLK:=bExe_Kill_Prog, Q=> );
CASE Exe_kill_step OF
	0:
		IF R_TRIG_Exekill.Q THEN
			NT_StartProcess_Kill.START:=FALSE;
			NT_StartProcess_Kill.PATHSTR:='C:\HZB\OpcIocShell\IDControlIOC\killcmd.bat';
			//NT_StartProcess_Kill.DIRNAME:='C:\Program Files (x86)\HZB\OpcIocShell\bin\opcIocShell.exe';
			Exe_kill_step:=10;
		END_IF;
	10:
		NT_StartProcess_Kill.START:=TRUE;
		Exe_kill_step:=20;
	20:
		IF NT_StartProcess_Kill.ERR THEN
			Exe_kill_step:=0;
		ELSE
			Exe_kill_step:=30;
		END_IF;

	30:
		NT_StartProcess_Kill.START:=TRUE;
		Exe_kill_step:=40;
	40:
		IF NOT NT_StartProcess_Kill.BUSY THEN
			NT_StartProcess_Kill.START:=FALSE;
			Exe_Kill_Done:=TRUE;
			Exe_kill_step:=0;
		END_IF;
END_CASE;

NT_StartProcess_Kill(
	NETID:='' ,
	PATHSTR:= ,
	DIRNAME:= , 
	COMNDLINE:= , 
	START:= ,
	ERRID=> );
END_ACTION

ACTION A_LEHeartBeatMonitor:
//monitor only while power on and not simulation or not use LE
IF NOT st_Power THEN
	RETURN;
END_IF
(**)
IF simulation THEN
	RETURN;
END_IF
IF NOT USELinearEncoder THEN
	RETURN;
END_IF

// 初始化
IF LEHeartBeatFirstScan THEN
    Velo_PhaseShifterLin_Last := PhaseShifterLin.NcToPlc.ActVelo;
    LEHeartBeatFirstScan := FALSE;
END_IF;

// 计算光栅前后速度差，速度差比位置差更敏感
DeltaVelo_PhaseShifterLin := ABS(PhaseShifterLin.NcToPlc.ActVelo - Velo_PhaseShifterLin_Last);
//PhaseShifter monitor
IF DeltaVelo_PhaseShifterLin > LEHeartBeatDeadZone THEN
    // 有变动，光栅正常，计数器归零，更新位置,重置所有状态
    StableTimer_PhaseShifterLin(IN := FALSE, PT := LEHeartBeatAlarmTime);
    Alarm_PhaseShifterLin := FALSE;
    Velo_PhaseShifterLin_Last := PhaseShifterLin.NcToPlc.ActVelo;  // 
    StableTime_PhaseShifterLin := T#0S;
	IsInitialPositionSet_PhaseShifter:=FALSE;
	Alarm_PhaseShifterMotorPos:=FALSE;
	Alarm_PhaseShifterMotorVelo:=FALSE;
ELSE
    //一点变动没有了，光栅异常，开始计时
    StableTimer_PhaseShifterLin(
        IN := TRUE,
        PT := LEHeartBeatAlarmTime,
        ET => StableTime_PhaseShifterLin
    );
	//记录电机初始位置，后后续对比做准备
	IF NOT IsInitialPositionSet_PhaseShifter THEN
        Pos_PhaseShifterMotor_Initial := Pos_PhaseShifterMotor;  // 记录初始位置
        IsInitialPositionSet_PhaseShifter := TRUE;
   	END_IF;
    
    // 100ms速度完全不变，开始监控电机速度和位置
    IF StableTimer_PhaseShifterLin.Q THEN
        Alarm_PhaseShifterLin := TRUE;  // 
			//电机位置对比及监测
			MotorPosChange_PhaseShifter:=ABS( Pos_PhaseShifterMotor-Pos_PhaseShifterMotor_Initial);
			IF MotorPosChange_PhaseShifter > Threshold_PhaseShifterMotorPos THEN
				Alarm_PhaseShifterMotorPos:=TRUE;
				ErrorID:=5001;
				ErrorDescription:='5001';
				Error:=TRUE;
				FB_PlcEmergencyStop();
				LED_Error:=TRUE;
			ELSE
				Alarm_PhaseShifterMotorPos:=FALSE;
			END_IF
			//电机速度监测
			IF Velo_PhaseShifterMotor > Threshold_PhaseShifterMotorVelo THEN
				Alarm_PhaseShifterMotorVelo:=TRUE;
				ErrorID:=5002;
				ErrorDescription:='5002';
				Error:=TRUE;
				FB_PlcEmergencyStop();
				LED_Error:=TRUE;
			ELSE
				Alarm_PhaseShifterMotorVelo:=FALSE;
			END_IF
    ELSE
        Alarm_PhaseShifterLin := FALSE;
	END_IF
END_IF
END_ACTION

ACTION A_LoadOpcIocShellExe:
R_TRIG_Exeload(CLK:=bExe_load_Prog, Q=> );
CASE Exe_load_step OF
	0:
		IF R_TRIG_Exeload.Q THEN
			NT_StartProcess_Load.START:=FALSE;
			NT_StartProcess_Load.PATHSTR:='C:\HZB\OpcIocShell\IDControlIOC\startTwinCATOPCServer.bat';
			Exe_load_step:=10;
		END_IF;
	10:
		NT_StartProcess_Load.START:=TRUE;
		Exe_load_step:=20;
	20:
		IF NT_StartProcess_Load.ERR THEN
			Exe_load_step:=0;
		ELSE
			Exe_load_step:=30;
		END_IF;
	30:
		IF NOT NT_StartProcess_Load.BUSY THEN
			NT_StartProcess_Load.START:=FALSE;
			Exe_Load_Done:=TRUE;
			Exe_load_step:=0;
		END_IF;
END_CASE;

NT_StartProcess_Load(
	NETID:='' ,
	PATHSTR:= ,
	DIRNAME:= , 
	COMNDLINE:= , 
	START:= ,
	ERRID=> );
END_ACTION

ACTION A_MonitorMotorAndLE:
//Monitoring Motor and LE Position/Velocity
IF 	ABS(DeltaPos_PhaseShifter) > ThresholdDeltaPos_PhaseShifter THEN
	ErrorID:=6001;
	Error:=TRUE;
	ErrorDescription:='ABS(DeltaPos_PhaseShifter) > ThresholdDeltaPos_PhaseShifter';
	FB_PlcEmergencyStop();
	LED_Error:=TRUE;
END_IF

IF ABS(DeltaVelo_PhaseShifter) > ThresholdDeltaVelo_PhaseShifter THEN
	ErrorID:=6002;
	Error:=TRUE;
	ErrorDescription:='ABS(DeltaVelo_PhaseShifter) > ThresholdDeltaVelo_PhaseShifter';
	FB_PlcEmergencyStop();
	LED_Error:=TRUE;
END_IF


(*
//
//IF NotMoving ,Threshold is less
//
IF NOT moveStatusLeftTop THEN
		IF 	ABS(DeltaPos_LeftTop) > ThresholdDeltaPos_LeftTop/3 THEN
		ErrorID:=6009;
		Error:=TRUE;
		ErrorDescription:='ABS(DeltaPos_LeftTop) > ThresholdDeltaPos_LeftTop/3';
		FB_PlcEmergencyStop();
		LED_Error:=TRUE;
	END_IF
END_IF
IF NOT moveStatusRightTop THEN
	IF ABS(DeltaPos_RightTop) > ThresholdDeltaPos_RightTop/3 THEN
		ErrorID:=6010;
		Error:=TRUE;
		ErrorDescription:='ABS(DeltaPos_RightTop) > ThresholdDeltaPos_RightTop/3';
		FB_PlcEmergencyStop();
		LED_Error:=TRUE;
	END_IF
END_IF
IF NOT moveStatusLeftBottom THEN
	IF ABS(DeltaPos_LeftBottom) > ThresholdDeltaPos_LeftBottom/3 THEN
		ErrorID:=6011;
		Error:=TRUE;
		ErrorDescription:='ABS(DeltaPos_LeftBottom) > ThresholdDeltaPos_LeftBottom/3';
		FB_PlcEmergencyStop();
		LED_Error:=TRUE;
	END_IF
END_IF
IF NOT moveStatusRightBottom THEN
	IF ABS(DeltaPos_RightBottom) > ThresholdDeltaPos_RightBottom/3 THEN
		ErrorID:=6012;
		Error:=TRUE;
		ErrorDescription:='ABS(DeltaPos_RightBottom) > ThresholdDeltaPos_RightBottom';
		FB_PlcEmergencyStop();
		LED_Error:=TRUE;
	END_IF
END_IF

//
IF NOT moveStatusLeftTop THEN
	IF ABS(DeltaVelo_LeftTop) > ThresholdDeltaVelo_LeftTop/3 THEN
		ErrorID:=6013;
		Error:=TRUE;
		ErrorDescription:='ABS(DeltaVelo_LeftTop) > ThresholdDeltaVelo_LeftTop/3';
		FB_PlcEmergencyStop();
		LED_Error:=TRUE;
	END_IF
END_IF
IF NOT moveStatusRightTop THEN
	IF ABS(DeltaVelo_RightTop) > ThresholdDeltaVelo_RightTop/3 THEN
		ErrorID:=6014;
		Error:=TRUE;
		ErrorDescription:='ABS(DeltaVelo_RightTop) > ThresholdDeltaVelo_RightTop/3';
		FB_PlcEmergencyStop();
		LED_Error:=TRUE;
	END_IF
END_IF
IF NOT moveStatusLeftBottom THEN
	IF ABS(DeltaVelo_LeftBottom) > ThresholdDeltaVelo_LeftBottom/3 THEN
		ErrorID:=6015;
		Error:=TRUE;
		ErrorDescription:='ABS(DeltaVelo_LeftBottom) > ThresholdDeltaVelo_LeftBottom/3';
		FB_PlcEmergencyStop();
		LED_Error:=TRUE;
	END_IF
END_IF
IF NOT moveStatusRightBottom THEN
	IF ABS(DeltaVelo_RightBottom) > ThresholdDeltaVelo_RightBottom/3 THEN
		ErrorID:=6016;
		Error:=TRUE;
		ErrorDescription:='ABS(DeltaVelo_RightBottom) > ThresholdDeltaVelo_RightBottom/3';
		FB_PlcEmergencyStop();
		LED_Error:=TRUE;
	END_IF
END_IF
*)
END_ACTION

ACTION A_PosDiffDetectiion:
IF ABS(PosDiff_PhaseShifterLin_actual)>PosDiff_PhaseShifterLin THEN
	ErrorID:=201;
	Error:=TRUE;
	ErrorDescription:='ABS(PosDiff_PhaseShifterLin_actual)>PosDiff_PhaseShifterLin';
	FB_PlcEmergencyStop();
	LED_Error:=TRUE;
END_IF
END_ACTION

ACTION A_RestartDrivers:
Relay_EL2624[0]:=btn_RestartDriver1;
Relay_EL2624[1]:=btn_RestartDriver2;
Relay_EL2624[2]:=btn_RestartDriver3;
Relay_EL2624[3]:=btn_RestartDriver4;
Relay_EL2624[4]:=btn_RestartDriver5;
Relay_EL2624[5]:=btn_RestartDriver6;
Relay_EL2624[6]:=btn_RestartDriver7;
Relay_EL2624[7]:=btn_RestartDriver8;
///
//1.上升沿触发，btn_RestartDrivers上升沿后，btn_RestartDriver1~8全部高电平
//2、3s后，Driver1~8全部恢复低电平
//3、恢复全部状态到初始
///
RestartDriver_RTRIG(CLK:=btn_RestartDriversAll);
IF RestartDriver_RTRIG.Q THEN
	RestartDriver_Triggered:=TRUE;
	RestartDriver_Done:=FALSE;
END_IF
IF RestartDriver_Triggered THEN
	CASE RestartDriver_State OF
		0:
			btn_RestartDriver1:=TRUE;
			btn_RestartDriver2:=TRUE;
			btn_RestartDriver3:=TRUE;
			btn_RestartDriver4:=TRUE;
			btn_RestartDriver5:=TRUE;
			btn_RestartDriver6:=TRUE;
			btn_RestartDriver7:=TRUE;
			btn_RestartDriver8:=TRUE;
			//计时开始
			RestartDriver_TON(PT:=T#10S);
			RestartDriver_TON.IN:=TRUE;
			IF RestartDriver_TON.Q THEN
				RestartDriver_State:=1;
			END_IF
		1:
			btn_RestartDriver1:=FALSE;
			btn_RestartDriver2:=FALSE;
			btn_RestartDriver3:=FALSE;
			btn_RestartDriver4:=FALSE;
			btn_RestartDriver5:=FALSE;
			btn_RestartDriver6:=FALSE;
			btn_RestartDriver7:=FALSE;
			btn_RestartDriver8:=FALSE;
			RestartDriver_State:=88;
		88:
			RestartDriver_TON.IN:=FALSE;
			btn_RestartDriversAll:=FALSE;
			RestartDriver_State:=0;
			RestartDriver_Triggered:=FALSE;
			RestartDriver_Done:=TRUE;
	END_CASE
END_IF
END_ACTION

ACTION A_RestartTC:
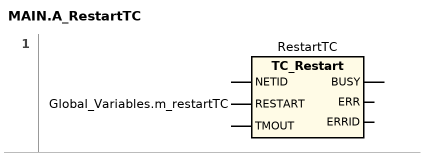
// NETWORK 1
RestartTC(RESTART := Global_Variables.m_restartTC); // TC_Restart
END_ACTION

ACTION A_SafePlcStartInit:
fb_ton0(PT:=t#1s);
fb_ton1(PT:=t#0.1s);
fb_ton2(PT:=t#0.1s);
fb_ton3(PT:=t#0.1s);

CASE SafeStatus OF
	0:
		IF COM_ERROR OR NOT Estop_Out THEN
			Err_Ack:=TRUE;
			fb_ton0.IN:=TRUE;
			SafeStatus:=1;
		ELSE
			SafePLCRunOK:=TRUE;
			SafeStatus:=0;
		END_IF
	1:
		IF fb_ton0.Q THEN
			Err_Ack:=FALSE;
			Safe_run:=TRUE;
			fb_ton1.IN:=TRUE;
			SafeStatus:=2;
		END_IF

	2:
		IF fb_ton1.Q THEN
			IF Estop_RunAndRestart=FALSE THEN
				Estop_RunAndRestart:=TRUE;
				fb_ton2.IN:=TRUE;
				SafeStatus:=3;
			END_IF
		END_IF
	3:
		IF fb_ton2.Q THEN
			IF Estop_RunAndRestart THEN
				Estop_RunAndRestart:=FALSE;
				fb_ton3.IN:=TRUE;
				SafeStatus:=4;
			END_IF
		END_IF
	4:
		IF fb_ton3.Q THEN
			IF Estop_Out THEN
				SafePLCRunOK:=TRUE;
				SafeStatus:=0;
			ELSE
				SafePLCRunOK:=FALSE;
				//Error:=TRUE;
				//ErrorId:=301;
				//ErrorDescription:='SafePLCRunOK fail';
			END_IF
		fb_ton0.IN:=FALSE;
		fb_ton1.IN:=FALSE;
		fb_ton2.IN:=FALSE;
		fb_ton3.IN:=FALSE;
		END_IF


END_CASE
END_ACTION

ACTION A_SetAxisPosition:
fb_ton4(PT:=t#0.5s);
CASE SetAxisPosState OF
	0:	(*FB_Set_AxisPosition*)
		FB_Set_AxisPosition(Execute:=TRUE);
		fb_ton4.IN:=TRUE;
		SetAxisPosState:=1;
	1:	(*wait*)
		FB_Set_AxisPosition();
		IF NOT FB_Set_AxisPosition.Done THEN		(*FB_Set_AxisPositionÃ»ÓÐÖ´ÐÐÍê£¬wait£¬³¬Ê±FB Error*)
			IF NOT fb_ton4.Q THEN
				SetAxisPosState:=1;
			ELSE
				SetAxisPosState:=99;
			END_IF
		ELSE
			SetAxisPosState:=88;
		END_IF
	88:
		SetAxisPosState:=0;
		SetAxisPositionDone:=TRUE;
		Error:=FALSE;
		ErrorID:=0;
		FB_Set_AxisPosition.Execute:=FALSE;
		fb_ton4.IN:=FALSE;
	99:
		SetAxisPosState:=99;
		SetAxisPositionDone:=FALSE;
		Error:=TRUE;
		FB_Set_AxisPosition.Execute:=FALSE;
		fb_ton4.IN:=FALSE;
		LED_Error:=TRUE;
		ErrorID:=401;
		ErrorDescription:='SetAxisPosition fail';
END_CASE
END_ACTION

ACTION A_SetLinearEncoderPositionBias:
//设置bias开始
A_SetLinearEncoderPositionBiasMC();
PositionBiasTON(PT:=T#0.1S);
CASE state_setLEPosBias OF
	0:
		PositionBiasTON.IN:=TRUE;
		IF MC_SetLEPosBias_PhaseShifter.Error THEN
			state_setLEPosBias:=-100;
		ELSE 
			state_setLEPosBias:=1;
		END_IF
	1:
		IF NOT MC_SetLEPosBias_PhaseShifter.Done  THEN
			MC_SetLEPosBias_PhaseShifter.Execute:=TRUE;
			state_setLEPosBias:=2;
		ELSE
			state_setLEPosBias:=-100;
		END_IF
	2:
		IF NOT MC_SetLEPosBias_PhaseShifter.Done THEN
			IF NOT PositionBiasTON.Q THEN
				state_setLEPosBias:=2;
			ELSE
				state_setLEPosBias:=-100;
			END_IF
		END_IF
		IF  MC_SetLEPosBias_PhaseShifter.Done THEN
			state_setLEPosBias:=88;
		END_IF	
		IF MC_SetLEPosBias_PhaseShifter.Error THEN
			state_setLEPosBias:=-100;
		END_IF 
		
	88:
		PositionBiasTON.IN:=FALSE;
		PositionBiasDone:=TRUE;
	-100:
		PositionBiasTON.IN:=FALSE;
		PositionBiasDone:=FALSE;
		Error:=TRUE;
		ErrorId:=901;
		ErrorDescription:='Set LinearEncoderPositionBias Error';
		Plc_EmergencyStop:=FALSE;
END_CASE
END_ACTION

ACTION A_SetLinearEncoderPositionBiasMC:
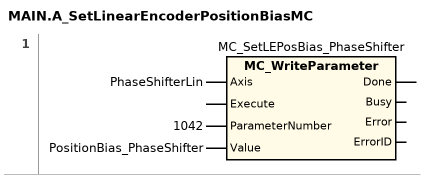
// NETWORK 1
MC_SetLEPosBias_PhaseShifter(
    Axis := PhaseShifterLin,
    ParameterNumber := 1042,
    Value := PositionBias_PhaseShifter); // MC_WriteParameter
END_ACTION

ACTION A_SetMotorAxisPosition:
fb_ton4_2(PT:=T#0.5S);
CASE SetMotorAxisPosState OF
	0:	(*FB_Set_AxisPosition*)
		FB_Set_MotorAxisPosition(Execute:=TRUE);
		fb_ton4_2.IN:=TRUE;
		SetMotorAxisPosState:=1;
	1:	(*wait*)
		FB_Set_MotorAxisPosition();
		IF NOT FB_Set_MotorAxisPosition.Done THEN		
			IF NOT fb_ton4_2.Q THEN
				SetMotorAxisPosState:=1;
			ELSE
				SetMotorAxisPosState:=99;
			END_IF
		ELSE
			SetMotorAxisPosState:=88;
		END_IF
	88:
		SetMotorAxisPosState:=0;
		SetMotorAxisPositionDone:=TRUE;
		Error:=FALSE;
		ErrorID:=0;
		FB_Set_MotorAxisPosition.Execute:=FALSE;
		fb_ton4_2.IN:=FALSE;
	99:
		SetMotorAxisPosState:=99;
		SetMotorAxisPositionDone:=FALSE;
		Error:=TRUE;
		FB_Set_MotorAxisPosition.Execute:=FALSE;
		fb_ton4.IN:=FALSE;
		LED_Error:=TRUE;
		ErrorID:=401;
		ErrorDescription:='SetMotorAxisPosition fail';
END_CASE
END_ACTION

END_PROGRAM
